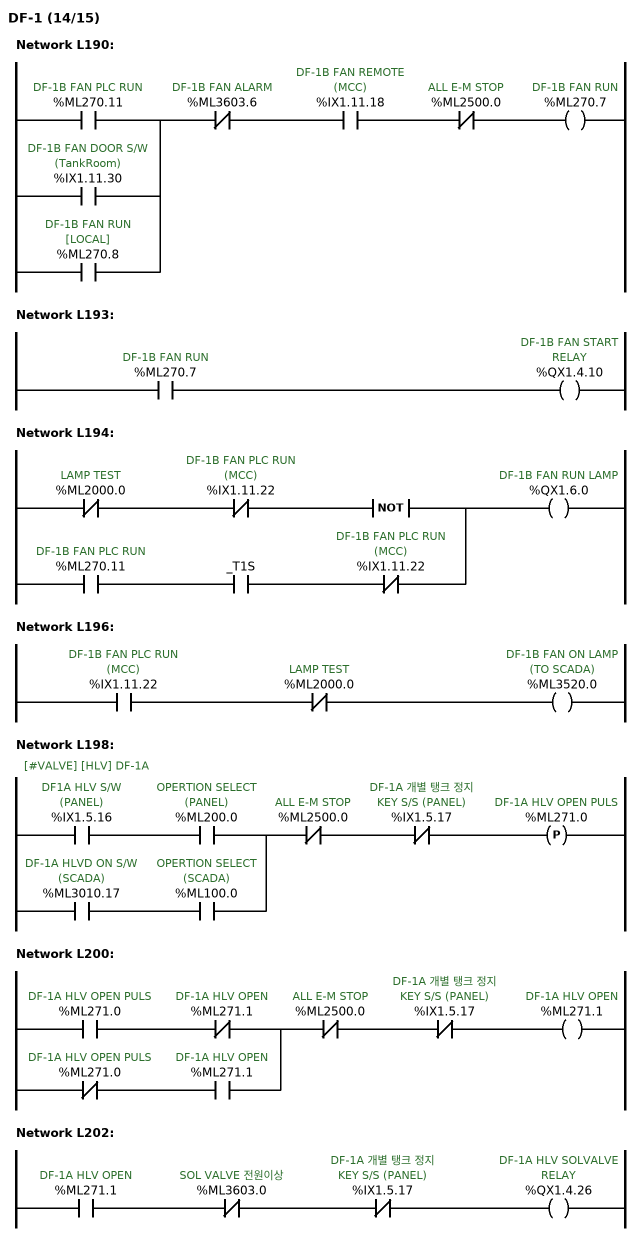
(* Rung L190 *)
%ML270.7 := (%ML270.11 OR %IX1.11.30 OR %ML270.8) AND NOT %ML3603.6 AND %IX1.11.18 AND NOT %ML2500.0;
(* Rung L193 *)
%QX1.4.10 := %ML270.7;
(* Rung L194 *)
%QX1.6.0 := NOT (NOT %ML2000.0 AND NOT %IX1.11.22) OR (%ML270.11 AND _T1S AND NOT %IX1.11.22);
(* Rung L196 *)
%ML3520.0 := %IX1.11.22 AND NOT %ML2000.0;
(* [#VALVE] [HLV] DF-1A *)
(* Rung L198 *)
_e3(CLK := ((%IX1.5.16 AND %ML200.0) OR (%ML3010.17 AND %ML100.0)) AND NOT %ML2500.0 AND NOT %IX1.5.17);
%ML271.0 := _e3.Q;
(* Rung L200 *)
%ML271.1 := ((%ML271.0 AND NOT %ML271.1) OR (NOT %ML271.0 AND %ML271.1)) AND NOT %ML2500.0 AND NOT %IX1.5.17;
(* Rung L202 *)
%QX1.4.26 := %ML271.1 AND NOT %ML3603.0 AND NOT %IX1.5.17;

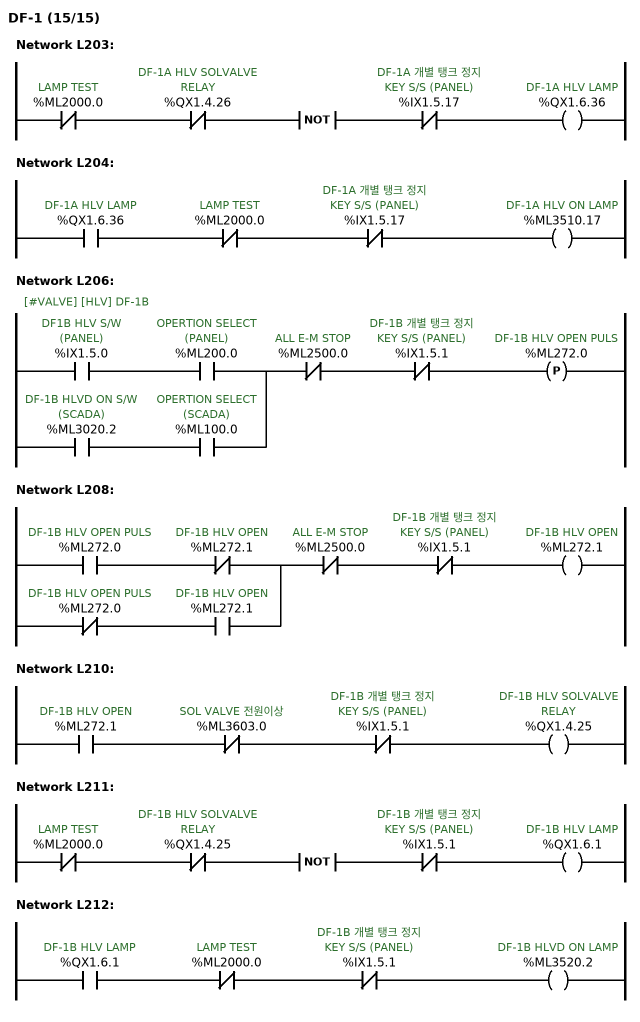
(* Rung L203 *)
%QX1.6.36 := NOT (NOT %ML2000.0 AND NOT %QX1.4.26) AND NOT %IX1.5.17;
(* Rung L204 *)
%ML3510.17 := %QX1.6.36 AND NOT %ML2000.0 AND NOT %IX1.5.17;
(* [#VALVE] [HLV] DF-1B *)
(* Rung L206 *)
_e4(CLK := ((%IX1.5.0 AND %ML200.0) OR (%ML3020.2 AND %ML100.0)) AND NOT %ML2500.0 AND NOT %IX1.5.1);
%ML272.0 := _e4.Q;
(* Rung L208 *)
%ML272.1 := ((%ML272.0 AND NOT %ML272.1) OR (NOT %ML272.0 AND %ML272.1)) AND NOT %ML2500.0 AND NOT %IX1.5.1;
(* Rung L210 *)
%QX1.4.25 := %ML272.1 AND NOT %ML3603.0 AND NOT %IX1.5.1;
(* Rung L211 *)
%QX1.6.1 := NOT (NOT %ML2000.0 AND NOT %QX1.4.25) AND NOT %IX1.5.1;
(* Rung L212 *)
%ML3520.2 := %QX1.6.1 AND NOT %ML2000.0 AND NOT %IX1.5.1;
END_PROGRAM

PROGRAM DF-M (* task: 스캔 프로그램 *)
VAR
    RP10 : TON;
    RP11 : TON;
    RP12 : TON;
    RP13 : TON;
    RP14 : TON;
    RP15 : TON;
    RP16 : TON;
    RP17 : TON;
    RP18 : TON;
    RP7 : TON;
    RP8 : TON;
    RP9 : TON;
    SUMP02 : TON; (* SP-2 *)
    SUMP04 : TON;
END_VAR
VAR
    _t1 : BOOL;
    _t2 : BOOL;
    _t3 : BOOL;
    _t4 : BOOL;
    _e5 : R_TRIG;
END_VAR

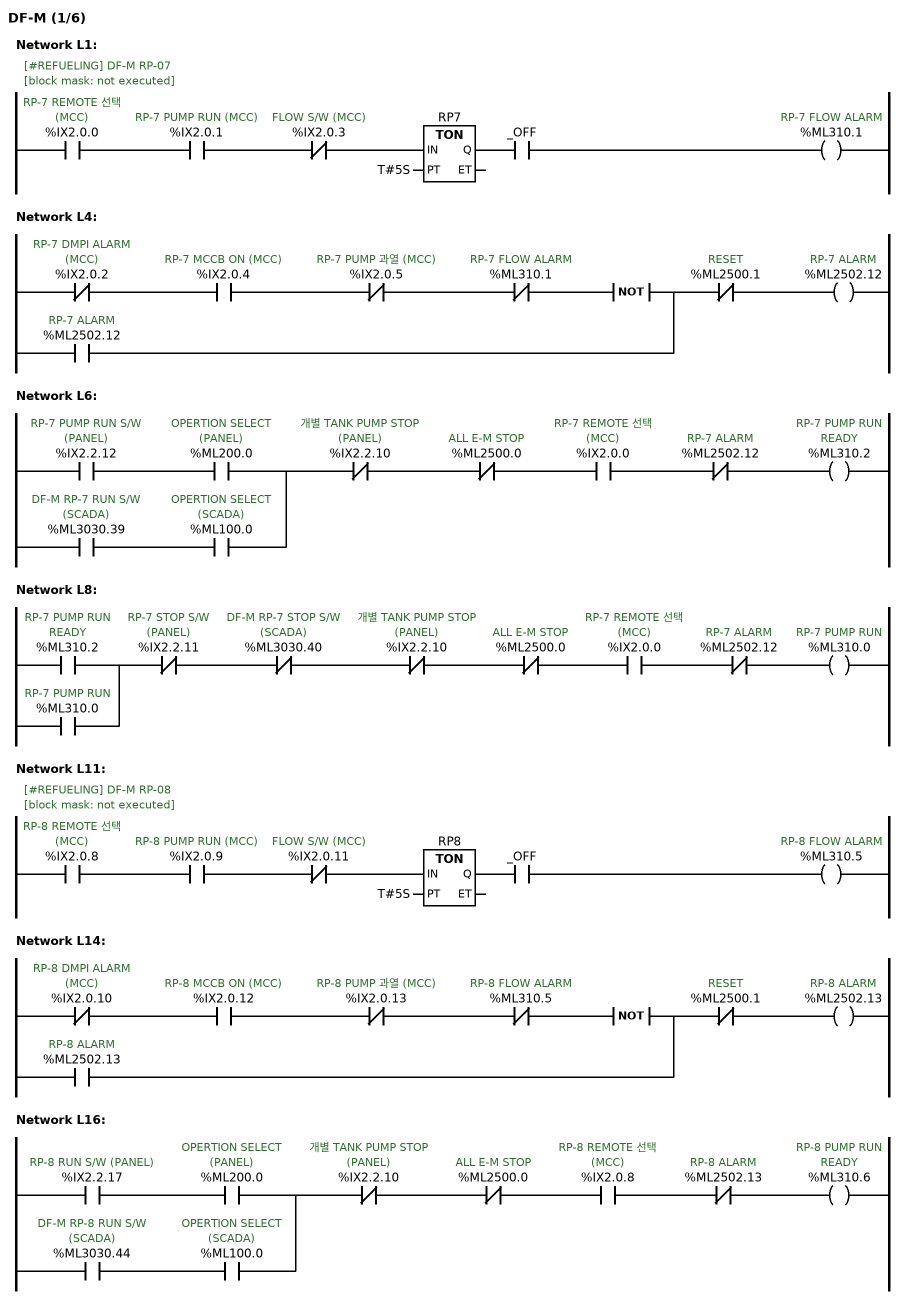
(* [#REFUELING] DF-M RP-07 *)
(* Rung L1 is block-masked: not executed *)
// RP7(IN := %IX2.0.0 AND %IX2.0.1 AND NOT %IX2.0.3, PT := T#5S);
// %ML310.1 := RP7.Q AND _OFF;
(* Rung L4 *)
%ML2502.12 := (NOT (NOT %IX2.0.2 AND %IX2.0.4 AND NOT %IX2.0.5 AND NOT %ML310.1) OR %ML2502.12) AND NOT %ML2500.1;
(* Rung L6 *)
%ML310.2 := ((%IX2.2.12 AND %ML200.0) OR (%ML3030.39 AND %ML100.0)) AND NOT %IX2.2.10 AND NOT %ML2500.0 AND %IX2.0.0 AND NOT %ML2502.12;
(* Rung L8 *)
%ML310.0 := (%ML310.2 OR %ML310.0) AND NOT %IX2.2.11 AND NOT %ML3030.40 AND NOT %IX2.2.10 AND NOT %ML2500.0 AND %IX2.0.0 AND NOT %ML2502.12;
(* [#REFUELING] DF-M RP-08 *)
(* Rung L11 is block-masked: not executed *)
// RP8(IN := %IX2.0.8 AND %IX2.0.9 AND NOT %IX2.0.11, PT := T#5S);
// %ML310.5 := RP8.Q AND _OFF;
(* Rung L14 *)
%ML2502.13 := (NOT (NOT %IX2.0.10 AND %IX2.0.12 AND NOT %IX2.0.13 AND NOT %ML310.5) OR %ML2502.13) AND NOT %ML2500.1;
(* Rung L16 *)
%ML310.6 := ((%IX2.2.17 AND %ML200.0) OR (%ML3030.44 AND %ML100.0)) AND NOT %IX2.2.10 AND NOT %ML2500.0 AND %IX2.0.8 AND NOT %ML2502.13;

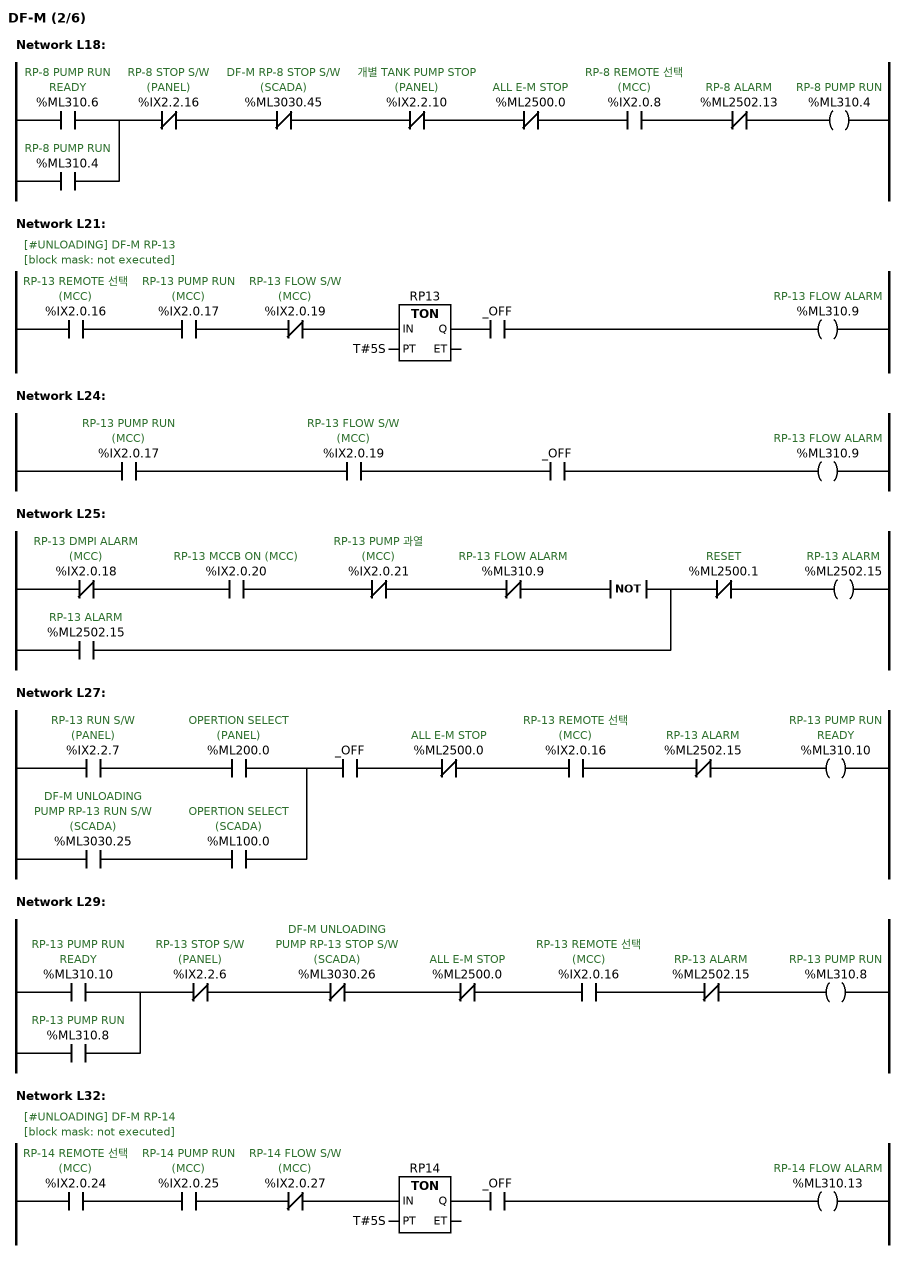
(* Rung L18 *)
%ML310.4 := (%ML310.6 OR %ML310.4) AND NOT %IX2.2.16 AND NOT %ML3030.45 AND NOT %IX2.2.10 AND NOT %ML2500.0 AND %IX2.0.8 AND NOT %ML2502.13;
(* [#UNLOADING] DF-M RP-13 *)
(* Rung L21 is block-masked: not executed *)
// RP13(IN := %IX2.0.16 AND %IX2.0.17 AND NOT %IX2.0.19, PT := T#5S);
// %ML310.9 := RP13.Q AND _OFF;
(* Rung L24 *)
%ML310.9 := %IX2.0.17 AND %IX2.0.19 AND _OFF;
(* Rung L25 *)
%ML2502.15 := (NOT (NOT %IX2.0.18 AND %IX2.0.20 AND NOT %IX2.0.21 AND NOT %ML310.9) OR %ML2502.15) AND NOT %ML2500.1;
(* Rung L27 *)
%ML310.10 := ((%IX2.2.7 AND %ML200.0) OR (%ML3030.25 AND %ML100.0)) AND _OFF AND NOT %ML2500.0 AND %IX2.0.16 AND NOT %ML2502.15;
(* Rung L29 *)
%ML310.8 := (%ML310.10 OR %ML310.8) AND NOT %IX2.2.6 AND NOT %ML3030.26 AND NOT %ML2500.0 AND %IX2.0.16 AND NOT %ML2502.15;
(* [#UNLOADING] DF-M RP-14 *)
(* Rung L32 is block-masked: not executed *)
// RP14(IN := %IX2.0.24 AND %IX2.0.25 AND NOT %IX2.0.27, PT := T#5S);
// %ML310.13 := RP14.Q AND _OFF;

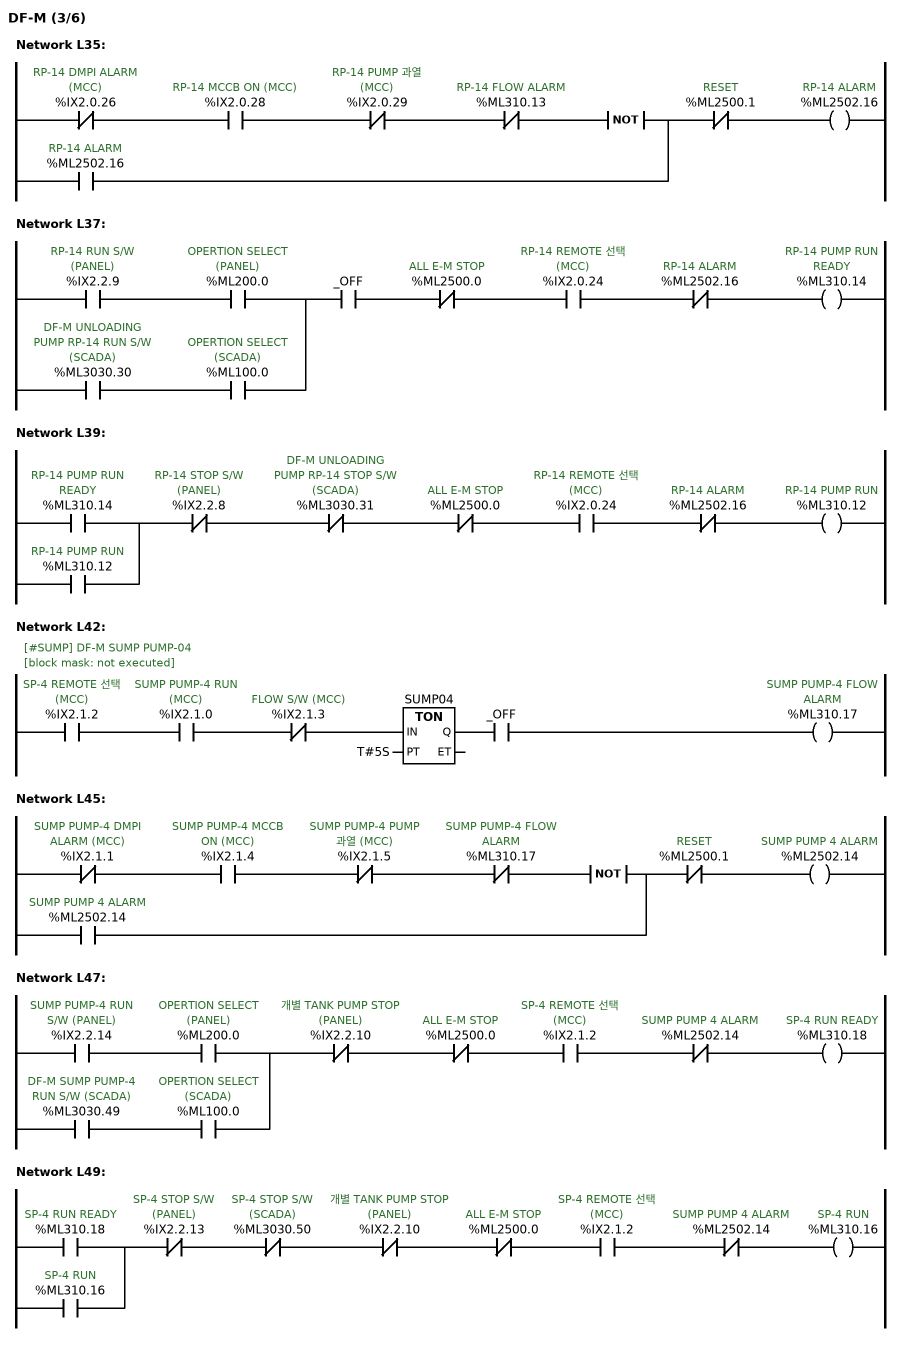
(* Rung L35 *)
%ML2502.16 := (NOT (NOT %IX2.0.26 AND %IX2.0.28 AND NOT %IX2.0.29 AND NOT %ML310.13) OR %ML2502.16) AND NOT %ML2500.1;
(* Rung L37 *)
%ML310.14 := ((%IX2.2.9 AND %ML200.0) OR (%ML3030.30 AND %ML100.0)) AND _OFF AND NOT %ML2500.0 AND %IX2.0.24 AND NOT %ML2502.16;
(* Rung L39 *)
%ML310.12 := (%ML310.14 OR %ML310.12) AND NOT %IX2.2.8 AND NOT %ML3030.31 AND NOT %ML2500.0 AND %IX2.0.24 AND NOT %ML2502.16;
(* [#SUMP] DF-M SUMP PUMP-04 *)
(* Rung L42 is block-masked: not executed *)
// SUMP04(IN := %IX2.1.2 AND %IX2.1.0 AND NOT %IX2.1.3, PT := T#5S);
// %ML310.17 := SUMP04.Q AND _OFF;
(* Rung L45 *)
%ML2502.14 := (NOT (NOT %IX2.1.1 AND %IX2.1.4 AND NOT %IX2.1.5 AND NOT %ML310.17) OR %ML2502.14) AND NOT %ML2500.1;
(* Rung L47 *)
%ML310.18 := ((%IX2.2.14 AND %ML200.0) OR (%ML3030.49 AND %ML100.0)) AND NOT %IX2.2.10 AND NOT %ML2500.0 AND %IX2.1.2 AND NOT %ML2502.14;
(* Rung L49 *)
%ML310.16 := (%ML310.18 OR %ML310.16) AND NOT %IX2.2.13 AND NOT %ML3030.50 AND NOT %IX2.2.10 AND NOT %ML2500.0 AND %IX2.1.2 AND NOT %ML2502.14;

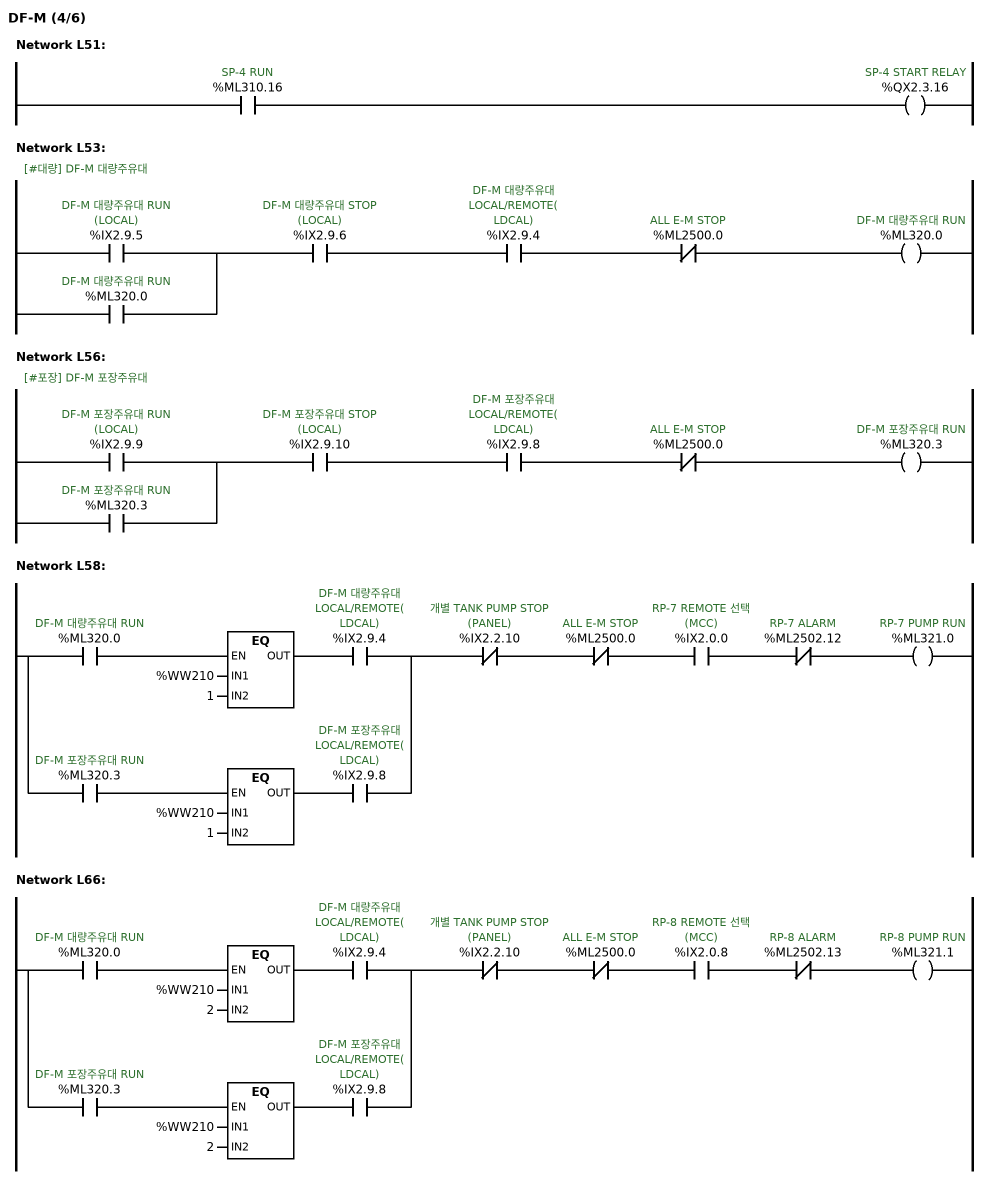
(* Rung L51 *)
%QX2.3.16 := %ML310.16;
(* [#대량] DF-M 대량주유대 *)
(* Rung L53 *)
%ML320.0 := (%IX2.9.5 OR %ML320.0) AND %IX2.9.6 AND %IX2.9.4 AND NOT %ML2500.0;
(* [#포장] DF-M 포장주유대 *)
(* Rung L56 *)
%ML320.3 := (%IX2.9.9 OR %ML320.3) AND %IX2.9.10 AND %IX2.9.8 AND NOT %ML2500.0;
(* Rung L58 *)
IF %ML320.0 THEN _t1 := %WW210 = 1; END_IF;
IF %ML320.3 THEN _t2 := %WW210 = 1; END_IF;
%ML321.0 := ((_t1 AND %IX2.9.4) OR (_t2 AND %IX2.9.8)) AND NOT %IX2.2.10 AND NOT %ML2500.0 AND %IX2.0.0 AND NOT %ML2502.12;
(* Rung L66 *)
IF %ML320.0 THEN _t3 := %WW210 = 2; END_IF;
IF %ML320.3 THEN _t4 := %WW210 = 2; END_IF;
%ML321.1 := ((_t3 AND %IX2.9.4) OR (_t4 AND %IX2.9.8)) AND NOT %IX2.2.10 AND NOT %ML2500.0 AND %IX2.0.8 AND NOT %ML2502.13;

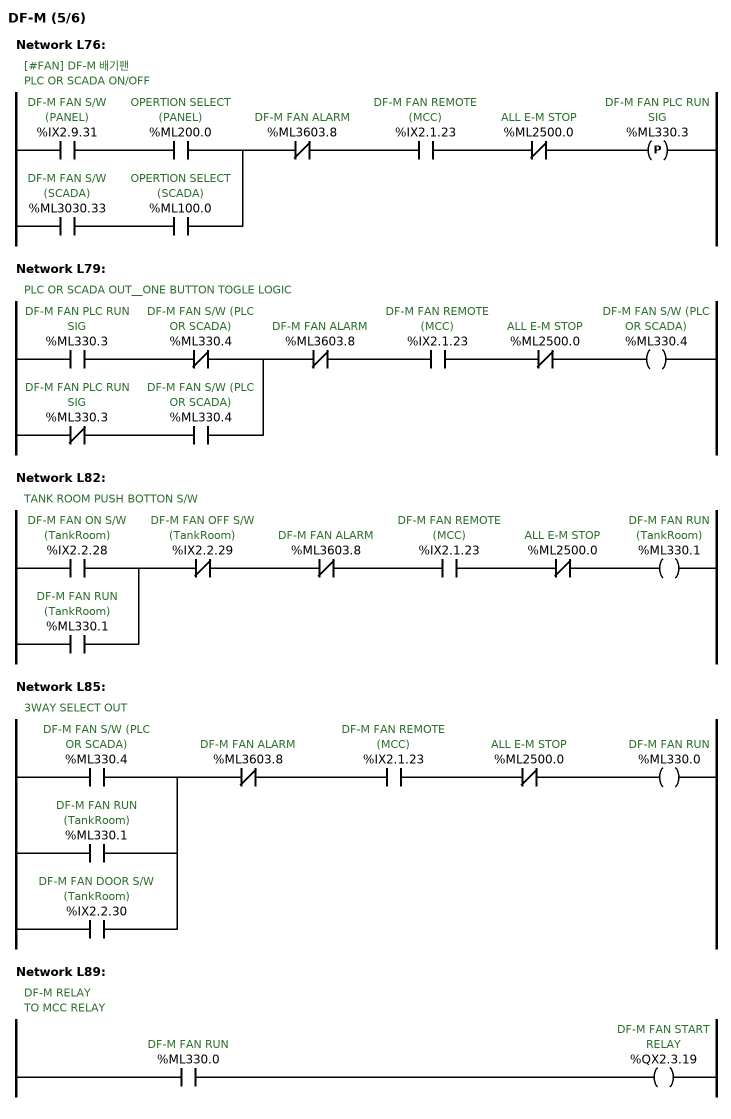
(* [#FAN] DF-M 배기팬 *)
(* PLC OR SCADA ON/OFF *)
(* Rung L76 *)
_e5(CLK := ((%IX2.9.31 AND %ML200.0) OR (%ML3030.33 AND %ML100.0)) AND NOT %ML3603.8 AND %IX2.1.23 AND NOT %ML2500.0);
%ML330.3 := _e5.Q;
(* PLC OR SCADA OUT__ONE BUTTON TOGLE LOGIC *)
(* Rung L79 *)
%ML330.4 := ((%ML330.3 AND NOT %ML330.4) OR (NOT %ML330.3 AND %ML330.4)) AND NOT %ML3603.8 AND %IX2.1.23 AND NOT %ML2500.0;
(* TANK ROOM PUSH BOTTON S/W *)
(* Rung L82 *)
%ML330.1 := (%IX2.2.28 OR %ML330.1) AND NOT %IX2.2.29 AND NOT %ML3603.8 AND %IX2.1.23 AND NOT %ML2500.0;
(* 3WAY SELECT OUT *)
(* Rung L85 *)
%ML330.0 := (%ML330.4 OR %ML330.1 OR %IX2.2.30) AND NOT %ML3603.8 AND %IX2.1.23 AND NOT %ML2500.0;
(* DF-M RELAY *)
(* Rung L89 *)
%QX2.3.19 := %ML330.0;
(* TO MCC RELAY *)

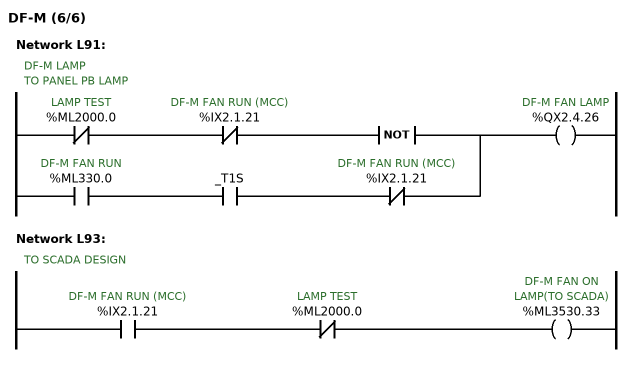
(* DF-M LAMP *)
(* Rung L91 *)
%QX2.4.26 := NOT (NOT %ML2000.0 AND NOT %IX2.1.21) OR (%ML330.0 AND _T1S AND NOT %IX2.1.21);
(* TO PANEL PB LAMP *)
(* Rung L93 *)
%ML3530.33 := %IX2.1.21 AND NOT %ML2000.0;
(* TO SCADA DESIGN *)
END_PROGRAM

PROGRAM MOGAS (* task: 스캔 프로그램 *)
VAR
    DP01 : TON; (* DRAIN PUMP FLOW SENSOR *)
    RP10 : TON;
    RP11 : TON;
    RP12 : TON;
    RP13 : TON;
    RP14 : TON;
    RP15 : TON;
    RP16 : TON;
    RP17 : TON;
    RP18 : TON;
    RP19 : TON;
    RP20 : TON;
    RP5 : TON;
    RP6 : TON;
    RP7 : TON;
    RP8 : TON;
    RP9 : TON;
    SUMP04 : TON;
END_VAR
VAR
    _t1 : BOOL;
    _t2 : BOOL;
    _t3 : BOOL;
    _t4 : BOOL;
    _e5 : R_TRIG;
END_VAR

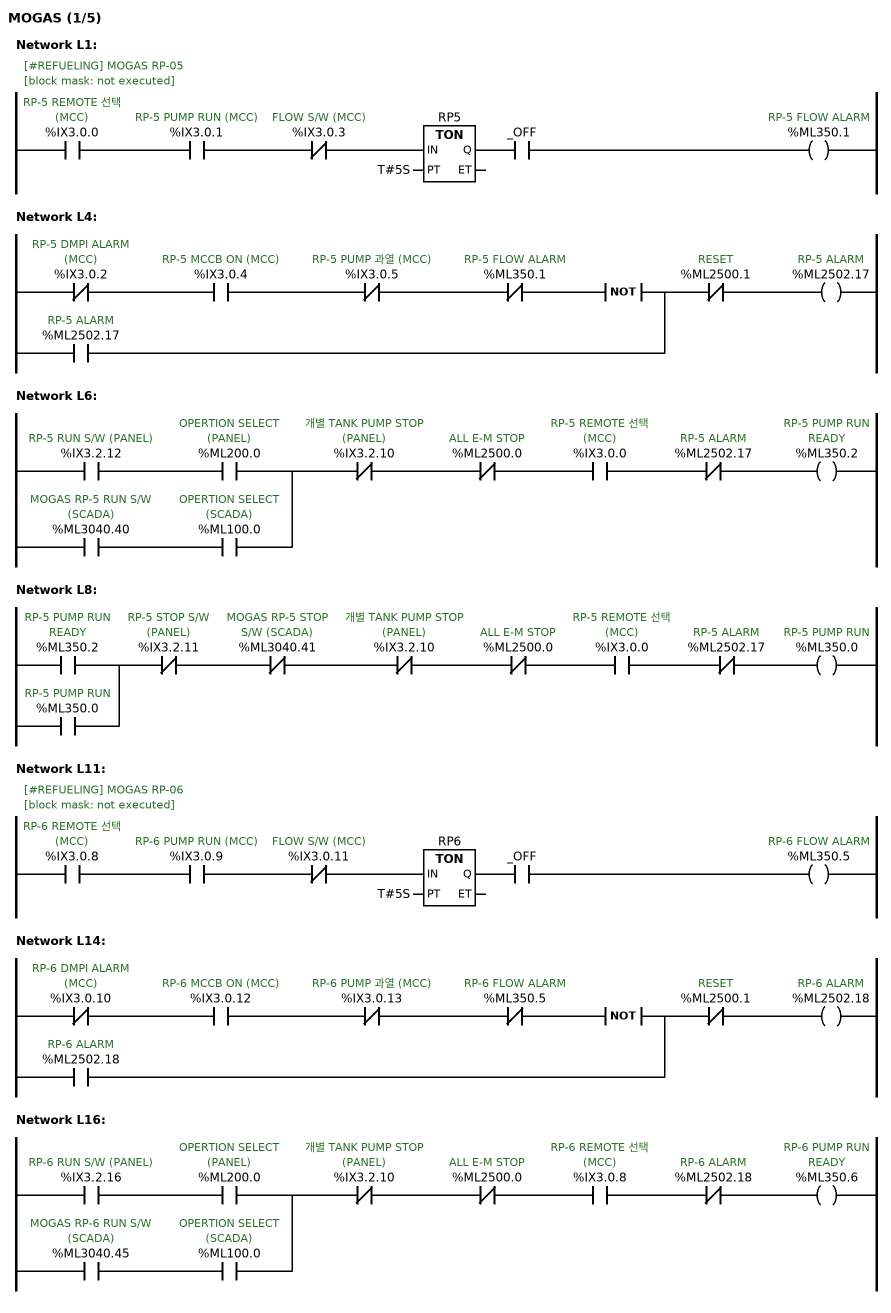
(* [#REFUELING] MOGAS RP-05 *)
(* Rung L1 is block-masked: not executed *)
// RP5(IN := %IX3.0.0 AND %IX3.0.1 AND NOT %IX3.0.3, PT := T#5S);
// %ML350.1 := RP5.Q AND _OFF;
(* Rung L4 *)
%ML2502.17 := (NOT (NOT %IX3.0.2 AND %IX3.0.4 AND NOT %IX3.0.5 AND NOT %ML350.1) OR %ML2502.17) AND NOT %ML2500.1;
(* Rung L6 *)
%ML350.2 := ((%IX3.2.12 AND %ML200.0) OR (%ML3040.40 AND %ML100.0)) AND NOT %IX3.2.10 AND NOT %ML2500.0 AND %IX3.0.0 AND NOT %ML2502.17;
(* Rung L8 *)
%ML350.0 := (%ML350.2 OR %ML350.0) AND NOT %IX3.2.11 AND NOT %ML3040.41 AND NOT %IX3.2.10 AND NOT %ML2500.0 AND %IX3.0.0 AND NOT %ML2502.17;
(* [#REFUELING] MOGAS RP-06 *)
(* Rung L11 is block-masked: not executed *)
// RP6(IN := %IX3.0.8 AND %IX3.0.9 AND NOT %IX3.0.11, PT := T#5S);
// %ML350.5 := RP6.Q AND _OFF;
(* Rung L14 *)
%ML2502.18 := (NOT (NOT %IX3.0.10 AND %IX3.0.12 AND NOT %IX3.0.13 AND NOT %ML350.5) OR %ML2502.18) AND NOT %ML2500.1;
(* Rung L16 *)
%ML350.6 := ((%IX3.2.16 AND %ML200.0) OR (%ML3040.45 AND %ML100.0)) AND NOT %IX3.2.10 AND NOT %ML2500.0 AND %IX3.0.8 AND NOT %ML2502.18;

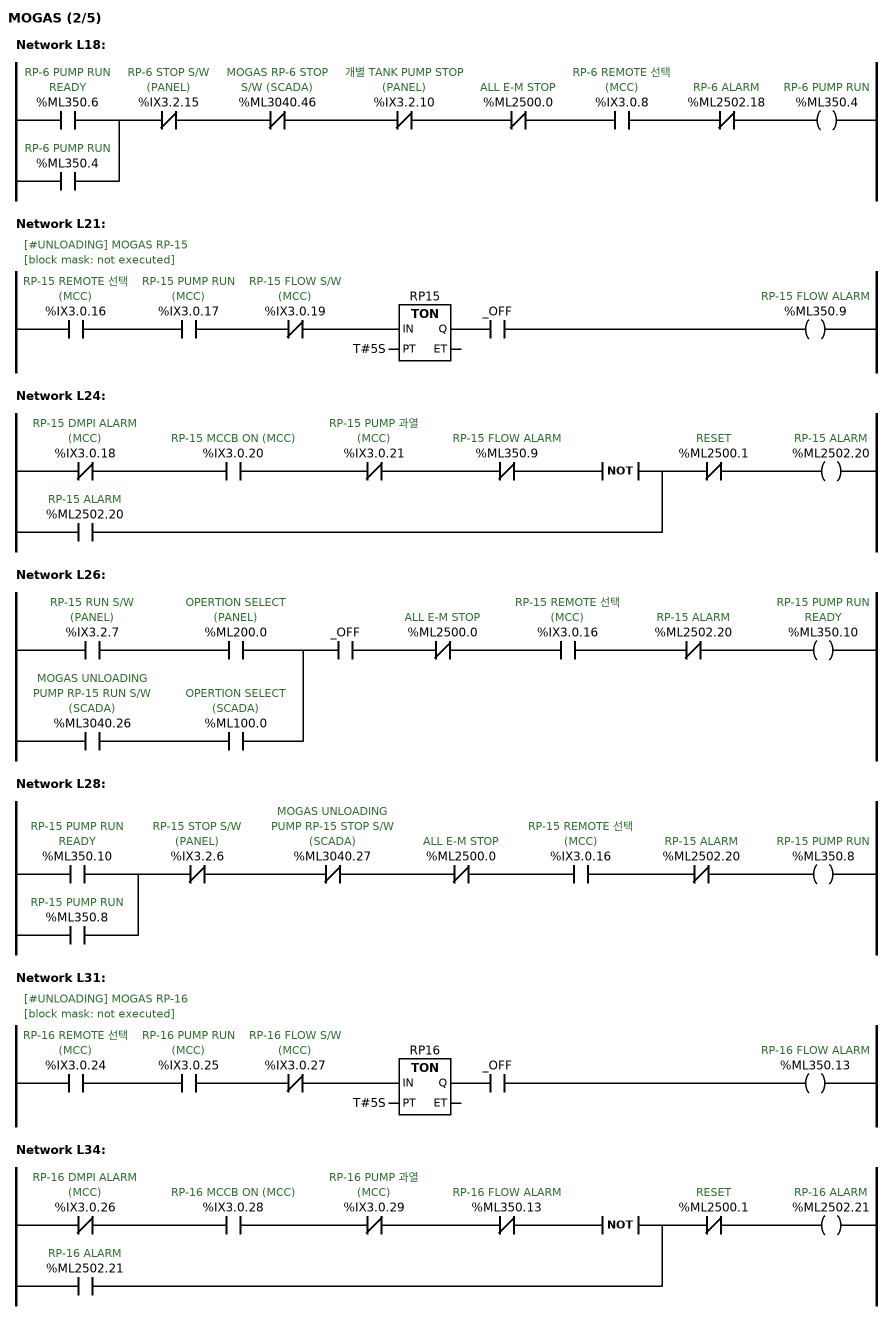
(* Rung L18 *)
%ML350.4 := (%ML350.6 OR %ML350.4) AND NOT %IX3.2.15 AND NOT %ML3040.46 AND NOT %IX3.2.10 AND NOT %ML2500.0 AND %IX3.0.8 AND NOT %ML2502.18;
(* [#UNLOADING] MOGAS RP-15 *)
(* Rung L21 is block-masked: not executed *)
// RP15(IN := %IX3.0.16 AND %IX3.0.17 AND NOT %IX3.0.19, PT := T#5S);
// %ML350.9 := RP15.Q AND _OFF;
(* Rung L24 *)
%ML2502.20 := (NOT (NOT %IX3.0.18 AND %IX3.0.20 AND NOT %IX3.0.21 AND NOT %ML350.9) OR %ML2502.20) AND NOT %ML2500.1;
(* Rung L26 *)
%ML350.10 := ((%IX3.2.7 AND %ML200.0) OR (%ML3040.26 AND %ML100.0)) AND _OFF AND NOT %ML2500.0 AND %IX3.0.16 AND NOT %ML2502.20;
(* Rung L28 *)
%ML350.8 := (%ML350.10 OR %ML350.8) AND NOT %IX3.2.6 AND NOT %ML3040.27 AND NOT %ML2500.0 AND %IX3.0.16 AND NOT %ML2502.20;
(* [#UNLOADING] MOGAS RP-16 *)
(* Rung L31 is block-masked: not executed *)
// RP16(IN := %IX3.0.24 AND %IX3.0.25 AND NOT %IX3.0.27, PT := T#5S);
// %ML350.13 := RP16.Q AND _OFF;
(* Rung L34 *)
%ML2502.21 := (NOT (NOT %IX3.0.26 AND %IX3.0.28 AND NOT %IX3.0.29 AND NOT %ML350.13) OR %ML2502.21) AND NOT %ML2500.1;

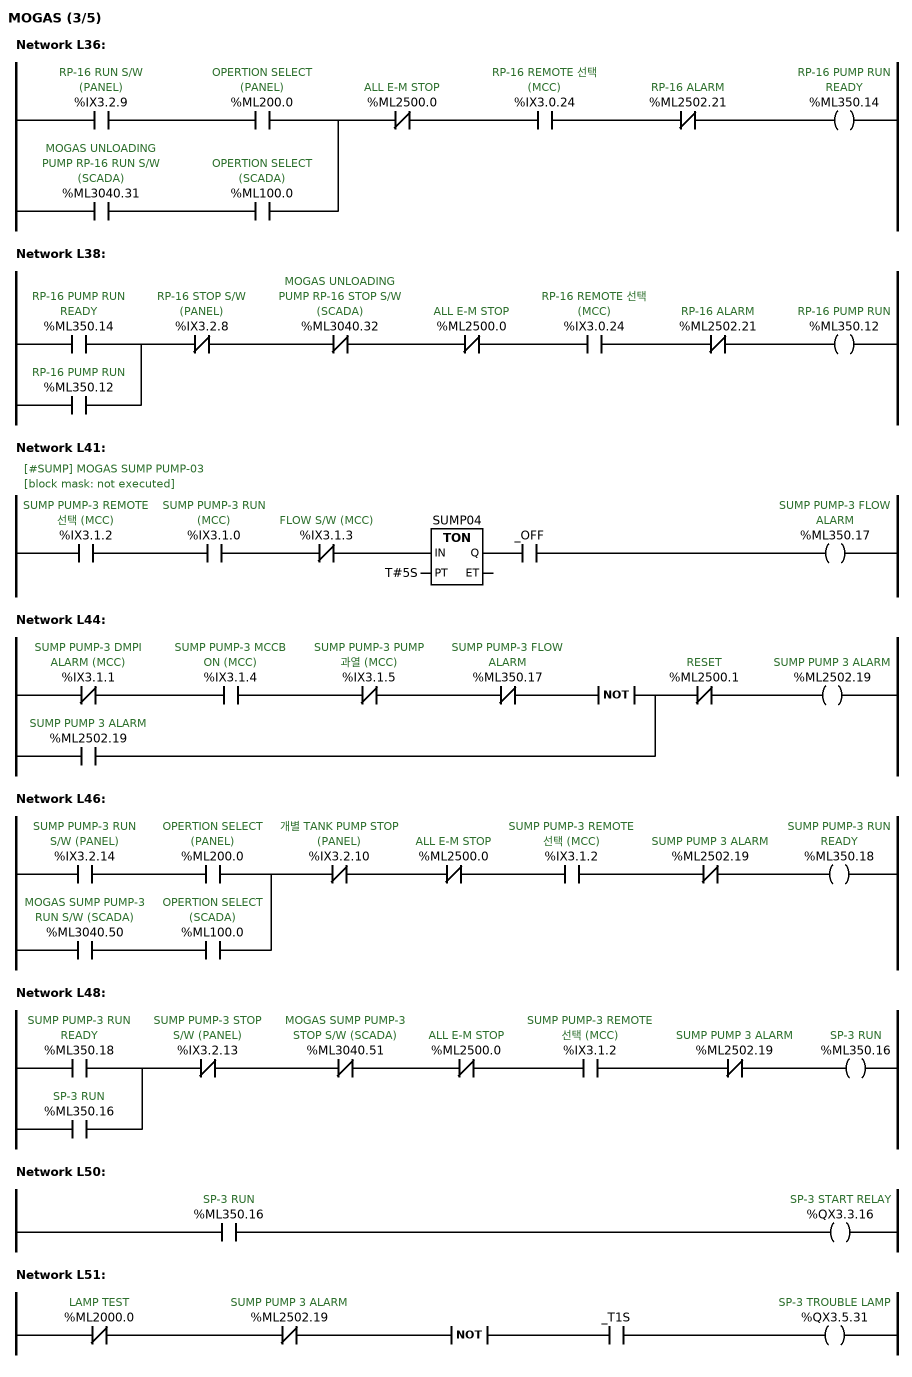
(* Rung L36 *)
%ML350.14 := ((%IX3.2.9 AND %ML200.0) OR (%ML3040.31 AND %ML100.0)) AND NOT %ML2500.0 AND %IX3.0.24 AND NOT %ML2502.21;
(* Rung L38 *)
%ML350.12 := (%ML350.14 OR %ML350.12) AND NOT %IX3.2.8 AND NOT %ML3040.32 AND NOT %ML2500.0 AND %IX3.0.24 AND NOT %ML2502.21;
(* [#SUMP] MOGAS SUMP PUMP-03 *)
(* Rung L41 is block-masked: not executed *)
// SUMP04(IN := %IX3.1.2 AND %IX3.1.0 AND NOT %IX3.1.3, PT := T#5S);
// %ML350.17 := SUMP04.Q AND _OFF;
(* Rung L44 *)
%ML2502.19 := (NOT (NOT %IX3.1.1 AND %IX3.1.4 AND NOT %IX3.1.5 AND NOT %ML350.17) OR %ML2502.19) AND NOT %ML2500.1;
(* Rung L46 *)
%ML350.18 := ((%IX3.2.14 AND %ML200.0) OR (%ML3040.50 AND %ML100.0)) AND NOT %IX3.2.10 AND NOT %ML2500.0 AND %IX3.1.2 AND NOT %ML2502.19;
(* Rung L48 *)
%ML350.16 := (%ML350.18 OR %ML350.16) AND NOT %IX3.2.13 AND NOT %ML3040.51 AND NOT %ML2500.0 AND %IX3.1.2 AND NOT %ML2502.19;
(* Rung L50 *)
%QX3.3.16 := %ML350.16;
(* Rung L51 *)
%QX3.5.31 := NOT (NOT %ML2000.0 AND NOT %ML2502.19) AND _T1S;

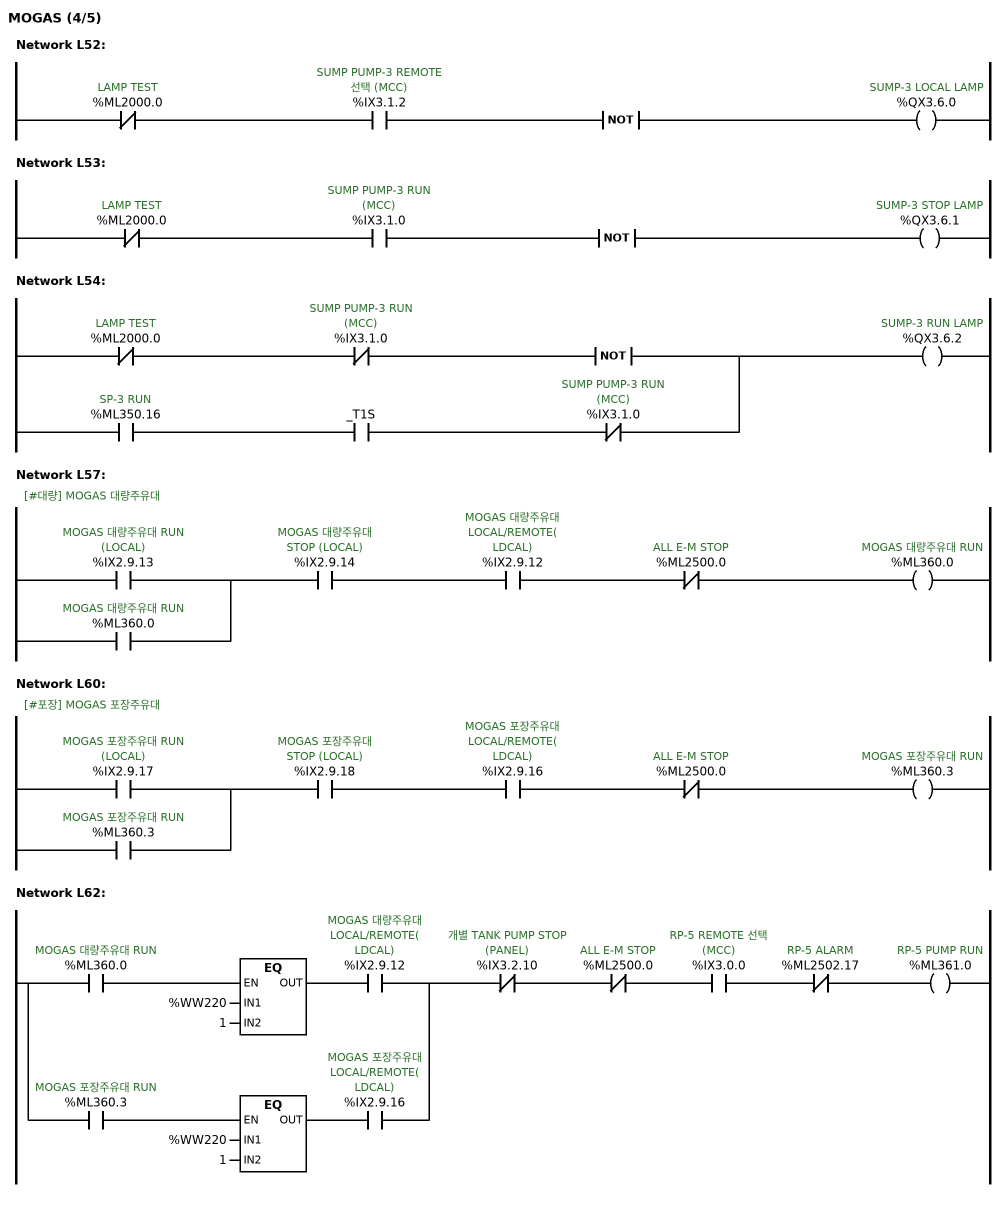
(* Rung L52 *)
%QX3.6.0 := NOT (NOT %ML2000.0 AND %IX3.1.2);
(* Rung L53 *)
%QX3.6.1 := NOT (NOT %ML2000.0 AND %IX3.1.0);
(* Rung L54 *)
%QX3.6.2 := NOT (NOT %ML2000.0 AND NOT %IX3.1.0) OR (%ML350.16 AND _T1S AND NOT %IX3.1.0);
(* [#대량] MOGAS 대량주유대 *)
(* Rung L57 *)
%ML360.0 := (%IX2.9.13 OR %ML360.0) AND %IX2.9.14 AND %IX2.9.12 AND NOT %ML2500.0;
(* [#포장] MOGAS 포장주유대 *)
(* Rung L60 *)
%ML360.3 := (%IX2.9.17 OR %ML360.3) AND %IX2.9.18 AND %IX2.9.16 AND NOT %ML2500.0;
(* Rung L62 *)
IF %ML360.0 THEN _t1 := %WW220 = 1; END_IF;
IF %ML360.3 THEN _t2 := %WW220 = 1; END_IF;
%ML361.0 := ((_t1 AND %IX2.9.12) OR (_t2 AND %IX2.9.16)) AND NOT %IX3.2.10 AND NOT %ML2500.0 AND %IX3.0.0 AND NOT %ML2502.17;

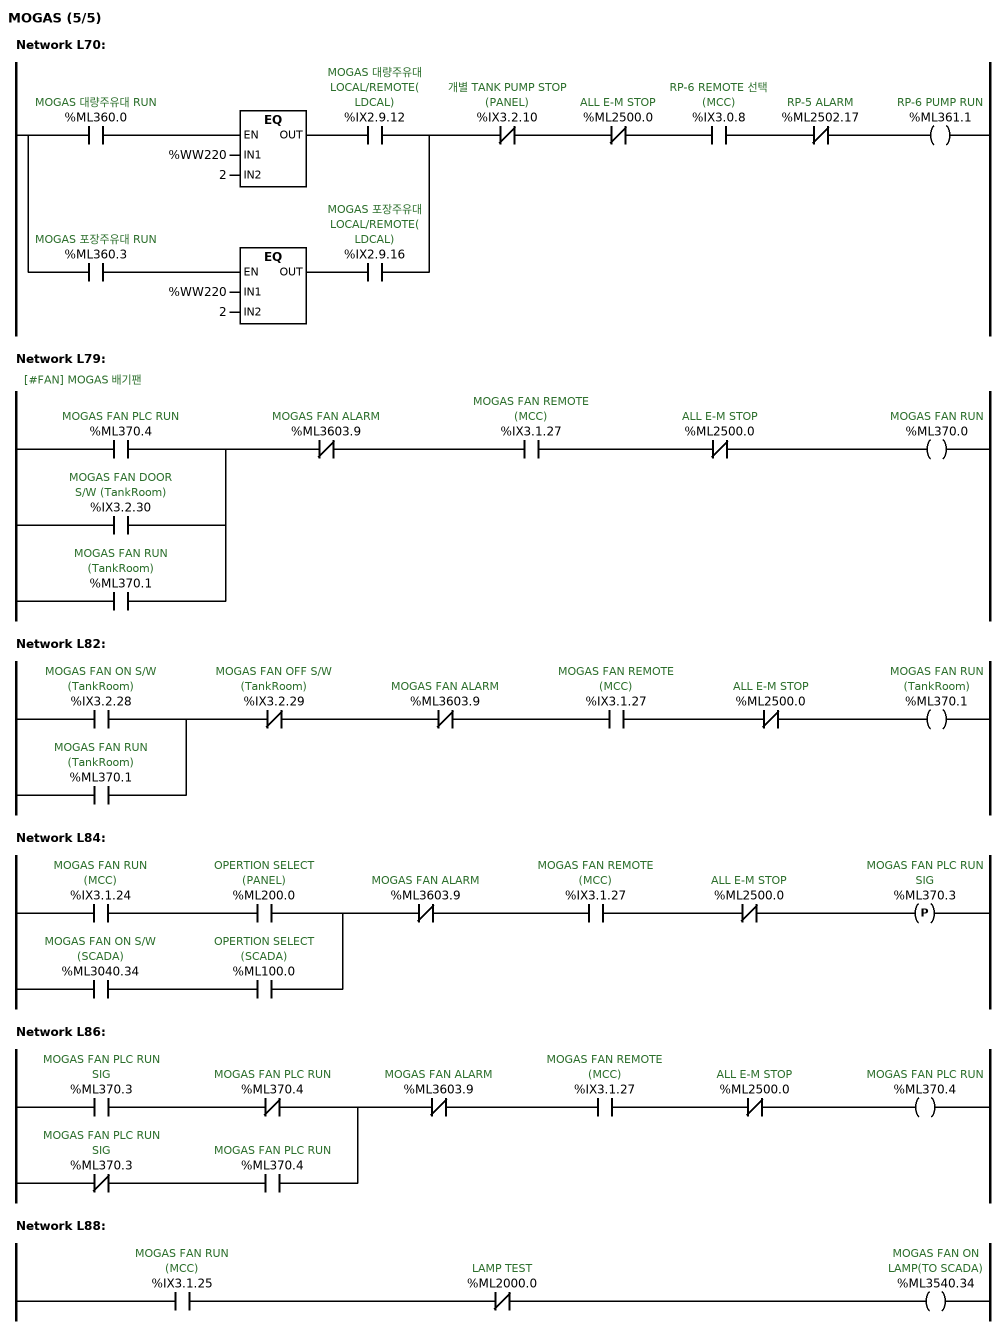
(* Rung L70 *)
IF %ML360.0 THEN _t3 := %WW220 = 2; END_IF;
IF %ML360.3 THEN _t4 := %WW220 = 2; END_IF;
%ML361.1 := ((_t3 AND %IX2.9.12) OR (_t4 AND %IX2.9.16)) AND NOT %IX3.2.10 AND NOT %ML2500.0 AND %IX3.0.8 AND NOT %ML2502.17;
(* [#FAN] MOGAS 배기팬 *)
(* Rung L79 *)
%ML370.0 := (%ML370.4 OR %IX3.2.30 OR %ML370.1) AND NOT %ML3603.9 AND %IX3.1.27 AND NOT %ML2500.0;
(* Rung L82 *)
%ML370.1 := (%IX3.2.28 OR %ML370.1) AND NOT %IX3.2.29 AND NOT %ML3603.9 AND %IX3.1.27 AND NOT %ML2500.0;
(* Rung L84 *)
_e5(CLK := ((%IX3.1.24 AND %ML200.0) OR (%ML3040.34 AND %ML100.0)) AND NOT %ML3603.9 AND %IX3.1.27 AND NOT %ML2500.0);
%ML370.3 := _e5.Q;
(* Rung L86 *)
%ML370.4 := ((%ML370.3 AND NOT %ML370.4) OR (NOT %ML370.3 AND %ML370.4)) AND NOT %ML3603.9 AND %IX3.1.27 AND NOT %ML2500.0;
(* Rung L88 *)
%ML3540.34 := %IX3.1.25 AND NOT %ML2000.0;
END_PROGRAM

PROGRAM ANALOGUE (* task: 스캔 프로그램 *)
VAR
    DF1A_LEVEL_PER : INT;
    DF1B_LEVEL_PER : INT;
    DFM_LEVEL_PER : INT;
    DTK1_LEVEL_PER : INT;
    DTK2_LEVEL_PER : INT;
    FIT_1 : INT;
    FIT_2 : INT;
    MOGAS_LEVEL_PER : INT;
END_VAR
VAR_EXTERNAL
    _0108_CH0_ACT : BOOL; (* AT %UX1.8.16 *) (* 절연형 아날로그입력 모듈: 채널0 운전중 *)
    _0108_CH0_DATA : INT; (* AT %UW1.8.2 *) (* 절연형 아날로그입력 모듈: 채널0 변환값 *)
    _0108_CH0_IDD : BOOL; (* AT %UX1.8.160 *) (* 절연형 아날로그입력 모듈: 채널0 입력단선검출 *)
    _0108_CH1_ACT : BOOL; (* AT %UX1.8.17 *) (* 절연형 아날로그입력 모듈: 채널1 운전중 *)
    _0108_CH1_DATA : INT; (* AT %UW1.8.3 *) (* 절연형 아날로그입력 모듈: 채널1 변환값 *)
    _0108_CH1_IDD : BOOL; (* AT %UX1.8.161 *) (* 절연형 아날로그입력 모듈: 채널1 입력단선검출 *)
    _0108_CH2_ACT : BOOL; (* AT %UX1.8.18 *) (* 절연형 아날로그입력 모듈: 채널2 운전중 *)
    _0108_CH2_DATA : INT; (* AT %UW1.8.4 *) (* 절연형 아날로그입력 모듈: 채널2 변환값 *)
    _0108_CH2_IDD : BOOL; (* AT %UX1.8.162 *) (* 절연형 아날로그입력 모듈: 채널2 입력단선검출 *)
    _0108_CH3_ACT : BOOL; (* AT %UX1.8.19 *) (* 절연형 아날로그입력 모듈: 채널3 운전중 *)
    _0108_CH3_DATA : INT; (* AT %UW1.8.5 *) (* 절연형 아날로그입력 모듈: 채널3 변환값 *)
    _0108_CH3_IDD : BOOL; (* AT %UX1.8.163 *) (* 절연형 아날로그입력 모듈: 채널3 입력단선검출 *)
    _0109_CH0_ACT : BOOL; (* AT %UX1.9.16 *) (* 절연형 아날로그출력 모듈: 채널0 운전중 *)
    _0109_CH0_DATA : INT; (* AT %UW1.9.3 *) (* 절연형 아날로그출력 모듈: 채널0 입력값 *)
    _0109_CH0_ERR : BOOL; (* AT %UX1.9.0 *) (* 절연형 아날로그출력 모듈: 채널0 에러 *)
    _0109_CH0_OUTEN : BOOL; (* AT %UX1.9.32 *) (* 절연형 아날로그출력 모듈: 채널0 출력상태설정 *)
    _0109_CH1_ACT : BOOL; (* AT %UX1.9.17 *) (* 절연형 아날로그출력 모듈: 채널1 운전중 *)
    _0109_CH1_DATA : INT; (* AT %UW1.9.4 *) (* 절연형 아날로그출력 모듈: 채널1 입력값 *)
    _0109_CH1_ERR : BOOL; (* AT %UX1.9.1 *) (* 절연형 아날로그출력 모듈: 채널1 에러 *)
    _0109_CH2_ACT : BOOL; (* AT %UX1.9.18 *) (* 절연형 아날로그출력 모듈: 채널2 운전중 *)
    _0109_CH2_DATA : INT; (* AT %UW1.9.5 *) (* 절연형 아날로그출력 모듈: 채널2 입력값 *)
    _0109_CH2_ERR : BOOL; (* AT %UX1.9.2 *) (* 절연형 아날로그출력 모듈: 채널2 에러 *)
    _0109_CH3_ACT : BOOL; (* AT %UX1.9.19 *) (* 절연형 아날로그출력 모듈: 채널3 운전중 *)
    _0109_CH3_DATA : INT; (* AT %UW1.9.6 *) (* 절연형 아날로그출력 모듈: 채널3 입력값 *)
    _0109_CH3_ERR : BOOL; (* AT %UX1.9.3 *) (* 절연형 아날로그출력 모듈: 채널3 에러 *)
    _0109_OUTEN : WORD; (* AT %UW1.9.2 *) (* 절연형 아날로그출력 모듈: 출력상태 설정 *)
    _0110_CH0_ACT : BOOL; (* AT %UX1.10.16 *) (* 절연형 아날로그출력 모듈: 채널0 운전중 *)
    _0110_CH0_DATA : INT; (* AT %UW1.10.3 *) (* 절연형 아날로그출력 모듈: 채널0 입력값 *)
    _0110_CH0_ERR : BOOL; (* AT %UX1.10.0 *) (* 절연형 아날로그출력 모듈: 채널0 에러 *)
    _0110_OUTEN : WORD; (* AT %UW1.10.2 *) (* 절연형 아날로그출력 모듈: 출력상태 설정 *)
    _0206_CH0_ACT : BOOL; (* AT %UX2.6.16 *) (* 절연형 아날로그입력 모듈: 채널0 운전중 *)
    _0206_CH0_DATA : INT; (* AT %UW2.6.2 *) (* 절연형 아날로그입력 모듈: 채널0 변환값 *)
    _0206_CH0_IDD : BOOL; (* AT %UX2.6.160 *) (* 절연형 아날로그입력 모듈: 채널0 입력단선검출 *)
    _0206_CH1_ACT : BOOL; (* AT %UX2.6.17 *) (* 절연형 아날로그입력 모듈: 채널1 운전중 *)
    _0206_CH1_DATA : INT; (* AT %UW2.6.3 *) (* 절연형 아날로그입력 모듈: 채널1 변환값 *)
    _0206_CH1_IDD : BOOL; (* AT %UX2.6.161 *) (* 절연형 아날로그입력 모듈: 채널1 입력단선검출 *)
    _0206_CH2_ACT : BOOL; (* AT %UX2.6.18 *) (* 절연형 아날로그입력 모듈: 채널2 운전중 *)
    _0206_CH2_DATA : INT; (* AT %UW2.6.4 *) (* 절연형 아날로그입력 모듈: 채널2 변환값 *)
    _0206_CH2_IDD : BOOL; (* AT %UX2.6.162 *) (* 절연형 아날로그입력 모듈: 채널2 입력단선검출 *)
    _0206_CH3_ACT : BOOL; (* AT %UX2.6.19 *) (* 절연형 아날로그입력 모듈: 채널3 운전중 *)
    _0206_CH3_DATA : INT; (* AT %UW2.6.5 *) (* 절연형 아날로그입력 모듈: 채널3 변환값 *)
    _0206_CH3_IDD : BOOL; (* AT %UX2.6.163 *) (* 절연형 아날로그입력 모듈: 채널3 입력단선검출 *)
    _0207_CH0_ACT : BOOL; (* AT %UX2.7.16 *) (* 절연형 아날로그출력 모듈: 채널0 운전중 *)
    _0207_CH0_DATA : INT; (* AT %UW2.7.3 *) (* 절연형 아날로그출력 모듈: 채널0 입력값 *)
    _0207_CH0_ERR : BOOL; (* AT %UX2.7.0 *) (* 절연형 아날로그출력 모듈: 채널0 에러 *)
    _0207_CH1_ACT : BOOL; (* AT %UX2.7.17 *) (* 절연형 아날로그출력 모듈: 채널1 운전중 *)
    _0207_CH1_DATA : INT; (* AT %UW2.7.4 *) (* 절연형 아날로그출력 모듈: 채널1 입력값 *)
    _0207_CH2_ACT : BOOL; (* AT %UX2.7.18 *) (* 절연형 아날로그출력 모듈: 채널2 운전중 *)
    _0207_CH2_DATA : INT; (* AT %UW2.7.5 *) (* 절연형 아날로그출력 모듈: 채널2 입력값 *)
    _0207_CH2_ERR : BOOL; (* AT %UX2.7.2 *) (* 절연형 아날로그출력 모듈: 채널2 에러 *)
    _0207_CH3_DATA : INT; (* AT %UW2.7.6 *) (* 절연형 아날로그출력 모듈: 채널3 입력값 *)
    _0207_OUTEN : WORD; (* AT %UW2.7.2 *) (* 절연형 아날로그출력 모듈: 출력상태 설정 *)
    _0307_CH0_ACT : BOOL; (* AT %UX3.7.16 *) (* 절연형 아날로그입력 모듈: 채널0 운전중 *)
    _0307_CH0_DATA : INT; (* AT %UW3.7.2 *) (* 절연형 아날로그입력 모듈: 채널0 변환값 *)
    _0307_CH0_IDD : BOOL; (* AT %UX3.7.160 *) (* 절연형 아날로그입력 모듈: 채널0 입력단선검출 *)
    _0307_CH1_ACT : BOOL; (* AT %UX3.7.17 *) (* 절연형 아날로그입력 모듈: 채널1 운전중 *)
    _0307_CH1_DATA : INT; (* AT %UW3.7.3 *) (* 절연형 아날로그입력 모듈: 채널1 변환값 *)
    _0307_CH1_IDD : BOOL; (* AT %UX3.7.161 *) (* 절연형 아날로그입력 모듈: 채널1 입력단선검출 *)
    _0307_CH2_ACT : BOOL; (* AT %UX3.7.18 *) (* 절연형 아날로그입력 모듈: 채널2 운전중 *)
    _0307_CH2_DATA : INT; (* AT %UW3.7.4 *) (* 절연형 아날로그입력 모듈: 채널2 변환값 *)
    _0307_CH2_IDD : BOOL; (* AT %UX3.7.162 *) (* 절연형 아날로그입력 모듈: 채널2 입력단선검출 *)
    _0307_CH3_DATA : INT; (* AT %UW3.7.5 *) (* 절연형 아날로그입력 모듈: 채널3 변환값 *)
    _0307_CH3_IDD : BOOL; (* AT %UX3.7.163 *) (* 절연형 아날로그입력 모듈: 채널3 입력단선검출 *)
    _0308_CH0_ACT : BOOL; (* AT %UX3.8.16 *) (* 절연형 아날로그출력 모듈: 채널0 운전중 *)
    _0308_CH0_DATA : INT; (* AT %UW3.8.3 *) (* 절연형 아날로그출력 모듈: 채널0 입력값 *)
    _0308_CH1_ACT : BOOL; (* AT %UX3.8.17 *) (* 절연형 아날로그출력 모듈: 채널1 운전중 *)
    _0308_CH1_DATA : INT; (* AT %UW3.8.4 *) (* 절연형 아날로그출력 모듈: 채널1 입력값 *)
    _0308_CH2_ACT : BOOL; (* AT %UX3.8.18 *) (* 절연형 아날로그출력 모듈: 채널2 운전중 *)
    _0308_CH2_DATA : INT; (* AT %UW3.8.5 *) (* 절연형 아날로그출력 모듈: 채널2 입력값 *)
    _0308_CH2_ERR : BOOL; (* AT %UX3.8.2 *) (* 절연형 아날로그출력 모듈: 채널2 에러 *)
    _0308_CH3_ACT : BOOL; (* AT %UX3.8.19 *) (* 절연형 아날로그출력 모듈: 채널3 운전중 *)
    _0308_CH3_DATA : INT; (* AT %UW3.8.6 *) (* 절연형 아날로그출력 모듈: 채널3 입력값 *)
    _0308_CH3_ERR : BOOL; (* AT %UX3.8.3 *) (* 절연형 아날로그출력 모듈: 채널3 에러 *)
    _0308_OUTEN : WORD; (* AT %UW3.8.2 *) (* 절연형 아날로그출력 모듈: 출력상태 설정 *)
END_VAR
VAR_EXTERNAL CONSTANT
    _F0308_CH0_DEC_RATE : UINT; (* 절연형 아날로그출력 모듈: 채널0 변화율 감소값 *)
    _F0308_CH0_STAT : UINT; (* 절연형 아날로그출력 모듈: 채널0 이상 상태 출력 설정값 *)
    _F0308_LIMIT_EN : UINT; (* 절연형 아날로그출력 모듈: 출력제한 채널 설정 *)
END_VAR
VAR
    _t1 : BOOL;
    _t2 : BOOL;
    _t3 : BOOL;
    _t4 : BOOL;
    _t5 : BOOL;
    _t6 : BOOL;
    _t7 : BOOL;
    _t8 : BOOL;
    _t9 : BOOL;
    _t10 : BOOL;
    _t11 : BOOL;
    _t12 : BOOL;
    _t13 : BOOL;
END_VAR

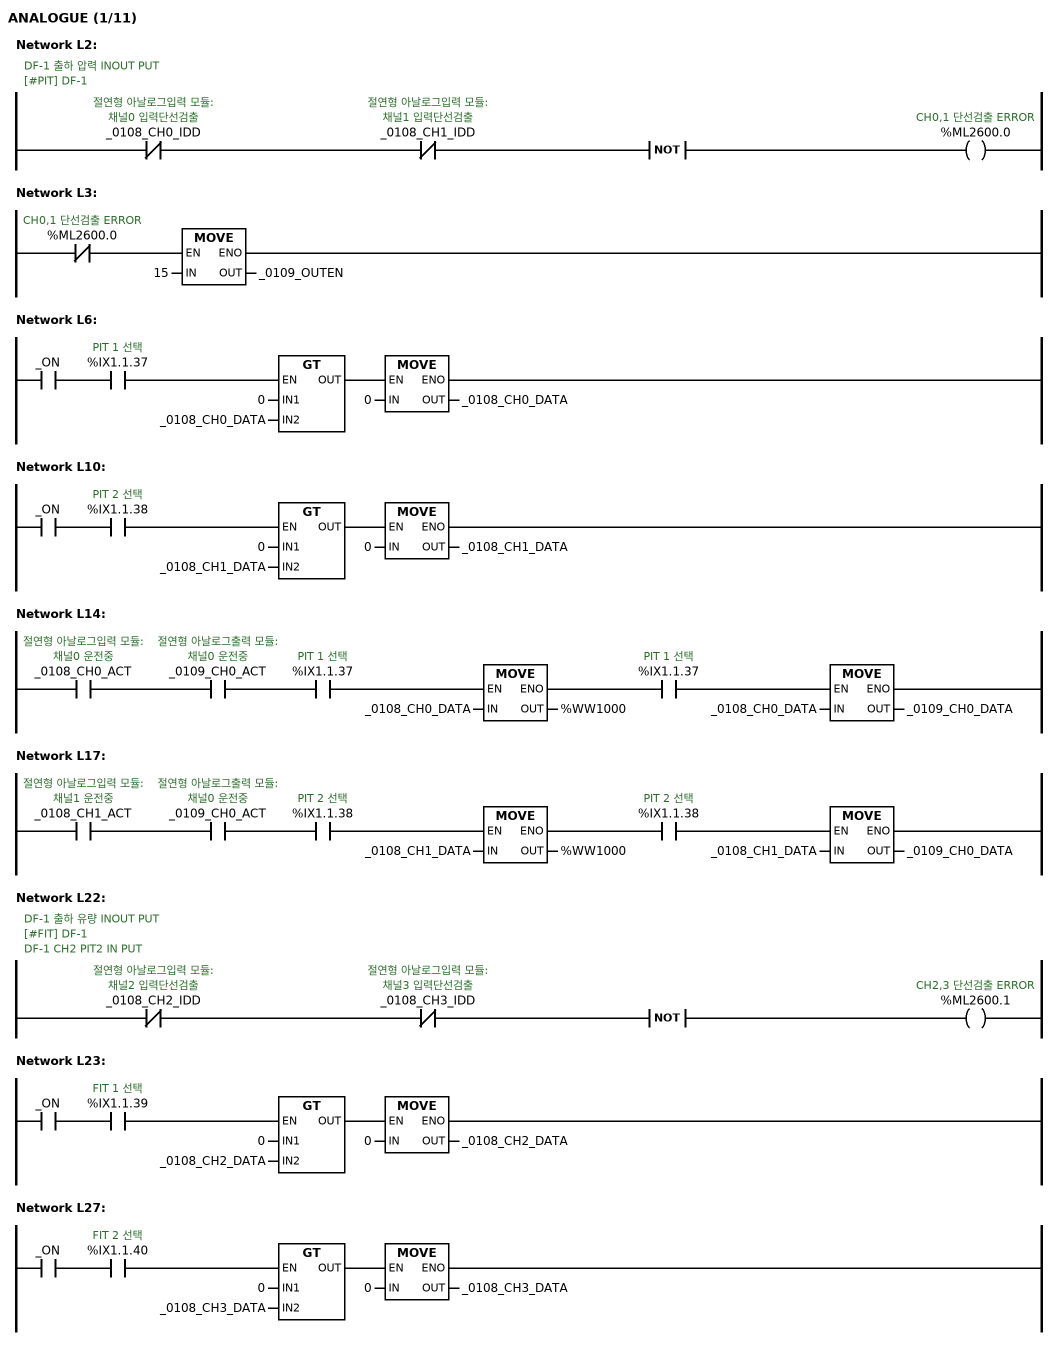
(* DF-1 출하 압력 INOUT PUT *)
(* [#PIT] DF-1 *)
(* Rung L2 *)
%ML2600.0 := NOT (NOT _0108_CH0_IDD AND NOT _0108_CH1_IDD);
(*  *)
(* Rung L3 *)
IF NOT %ML2600.0 THEN _0109_OUTEN := 15; END_IF;
(* Rung L6 *)
IF _ON AND %IX1.1.37 THEN _t1 := 0 > _0108_CH0_DATA; END_IF;
IF _t1 THEN _0108_CH0_DATA := 0; END_IF;
(* Rung L10 *)
IF _ON AND %IX1.1.38 THEN _t2 := 0 > _0108_CH1_DATA; END_IF;
IF _t2 THEN _0108_CH1_DATA := 0; END_IF;
(* Rung L14 *)
IF _0108_CH0_ACT AND _0109_CH0_ACT AND %IX1.1.37 THEN %WW1000 := _0108_CH0_DATA; END_IF;
IF _0108_CH0_ACT AND _0109_CH0_ACT AND %IX1.1.37 AND %IX1.1.37 THEN
    _0109_CH0_DATA := _0108_CH0_DATA;
END_IF;
(* Rung L17 *)
IF _0108_CH1_ACT AND _0109_CH0_ACT AND %IX1.1.38 THEN %WW1000 := _0108_CH1_DATA; END_IF;
IF _0108_CH1_ACT AND _0109_CH0_ACT AND %IX1.1.38 AND %IX1.1.38 THEN
    _0109_CH0_DATA := _0108_CH1_DATA;
END_IF;
(* DF-1 출하 유량 INOUT PUT *)
(* [#FIT] DF-1 *)
(* Rung L22 *)
%ML2600.1 := NOT (NOT _0108_CH2_IDD AND NOT _0108_CH3_IDD);
(* DF-1 CH2 PIT2 IN PUT *)
(* Rung L23 *)
IF _ON AND %IX1.1.39 THEN _t3 := 0 > _0108_CH2_DATA; END_IF;
IF _t3 THEN _0108_CH2_DATA := 0; END_IF;
(* Rung L27 *)
IF _ON AND %IX1.1.40 THEN _t4 := 0 > _0108_CH3_DATA; END_IF;
IF _t4 THEN _0108_CH3_DATA := 0; END_IF;

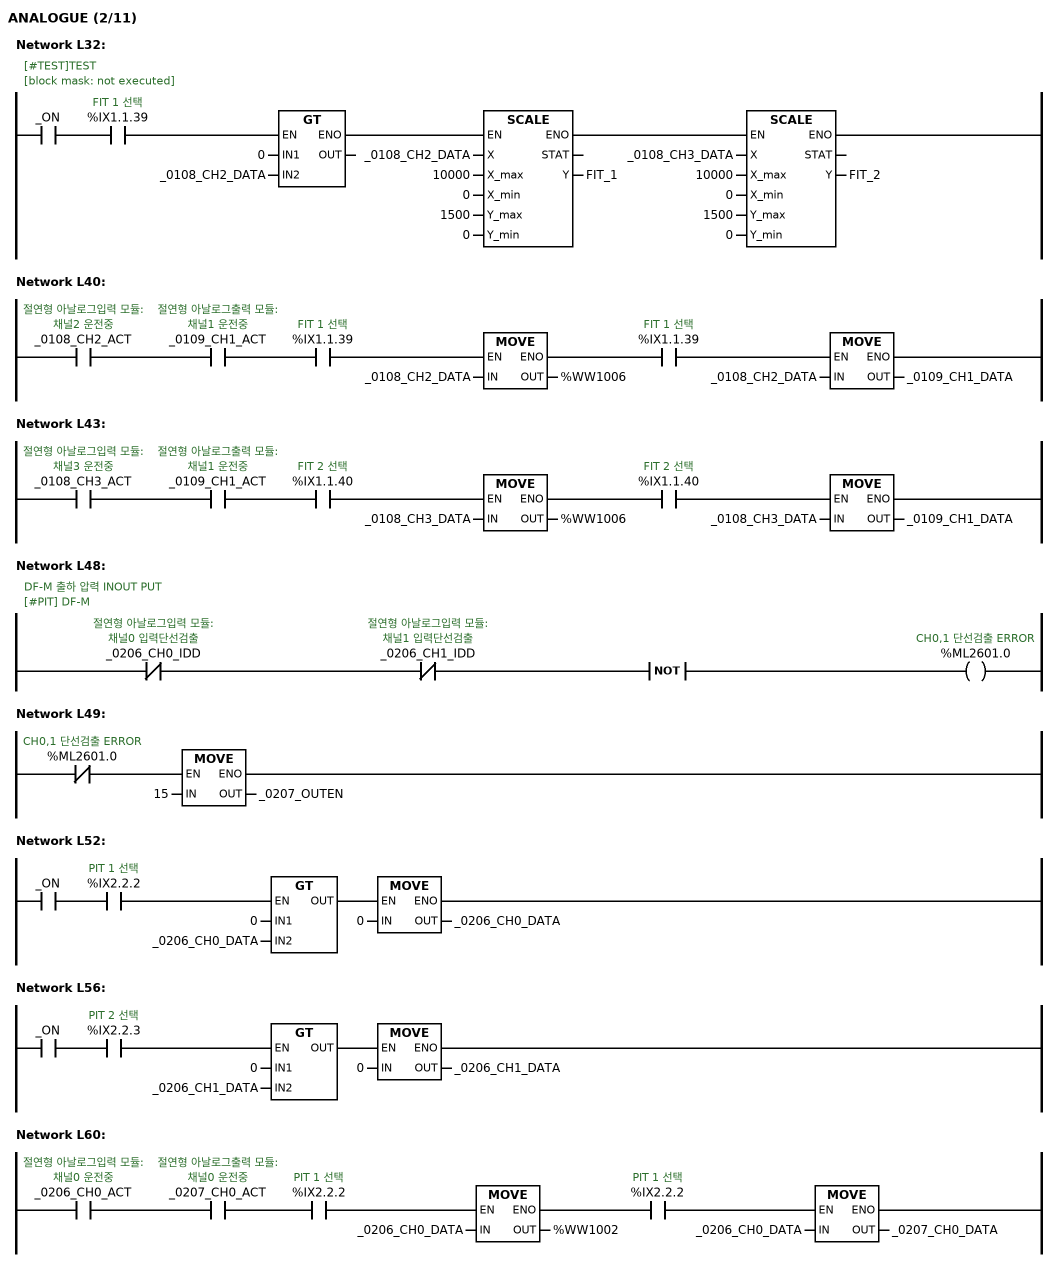
(* [#TEST]TEST *)
(* Rung L32 is block-masked: not executed *)
// IF _ON AND %IX1.1.39 THEN
//     _t5 := 0 > _0108_CH2_DATA;
//     SCALE(X := _0108_CH2_DATA, X_max := 10000, X_min := 0, Y_max := 1500, Y_min := 0, Y => FIT_1);
//     SCALE(X := _0108_CH3_DATA, X_max := 10000, X_min := 0, Y_max := 1500, Y_min := 0, Y => FIT_2);
// END_IF;
(*  *)
(* Rung L40 *)
IF _0108_CH2_ACT AND _0109_CH1_ACT AND %IX1.1.39 THEN %WW1006 := _0108_CH2_DATA; END_IF;
IF _0108_CH2_ACT AND _0109_CH1_ACT AND %IX1.1.39 AND %IX1.1.39 THEN
    _0109_CH1_DATA := _0108_CH2_DATA;
END_IF;
(* Rung L43 *)
IF _0108_CH3_ACT AND _0109_CH1_ACT AND %IX1.1.40 THEN %WW1006 := _0108_CH3_DATA; END_IF;
IF _0108_CH3_ACT AND _0109_CH1_ACT AND %IX1.1.40 AND %IX1.1.40 THEN
    _0109_CH1_DATA := _0108_CH3_DATA;
END_IF;
(* DF-M 출하 압력 INOUT PUT *)
(* [#PIT] DF-M *)
(* Rung L48 *)
%ML2601.0 := NOT (NOT _0206_CH0_IDD AND NOT _0206_CH1_IDD);
(*  *)
(* Rung L49 *)
IF NOT %ML2601.0 THEN _0207_OUTEN := 15; END_IF;
(* Rung L52 *)
IF _ON AND %IX2.2.2 THEN _t6 := 0 > _0206_CH0_DATA; END_IF;
IF _t6 THEN _0206_CH0_DATA := 0; END_IF;
(* Rung L56 *)
IF _ON AND %IX2.2.3 THEN _t7 := 0 > _0206_CH1_DATA; END_IF;
IF _t7 THEN _0206_CH1_DATA := 0; END_IF;
(* Rung L60 *)
IF _0206_CH0_ACT AND _0207_CH0_ACT AND %IX2.2.2 THEN %WW1002 := _0206_CH0_DATA; END_IF;
IF _0206_CH0_ACT AND _0207_CH0_ACT AND %IX2.2.2 AND %IX2.2.2 THEN
    _0207_CH0_DATA := _0206_CH0_DATA;
END_IF;

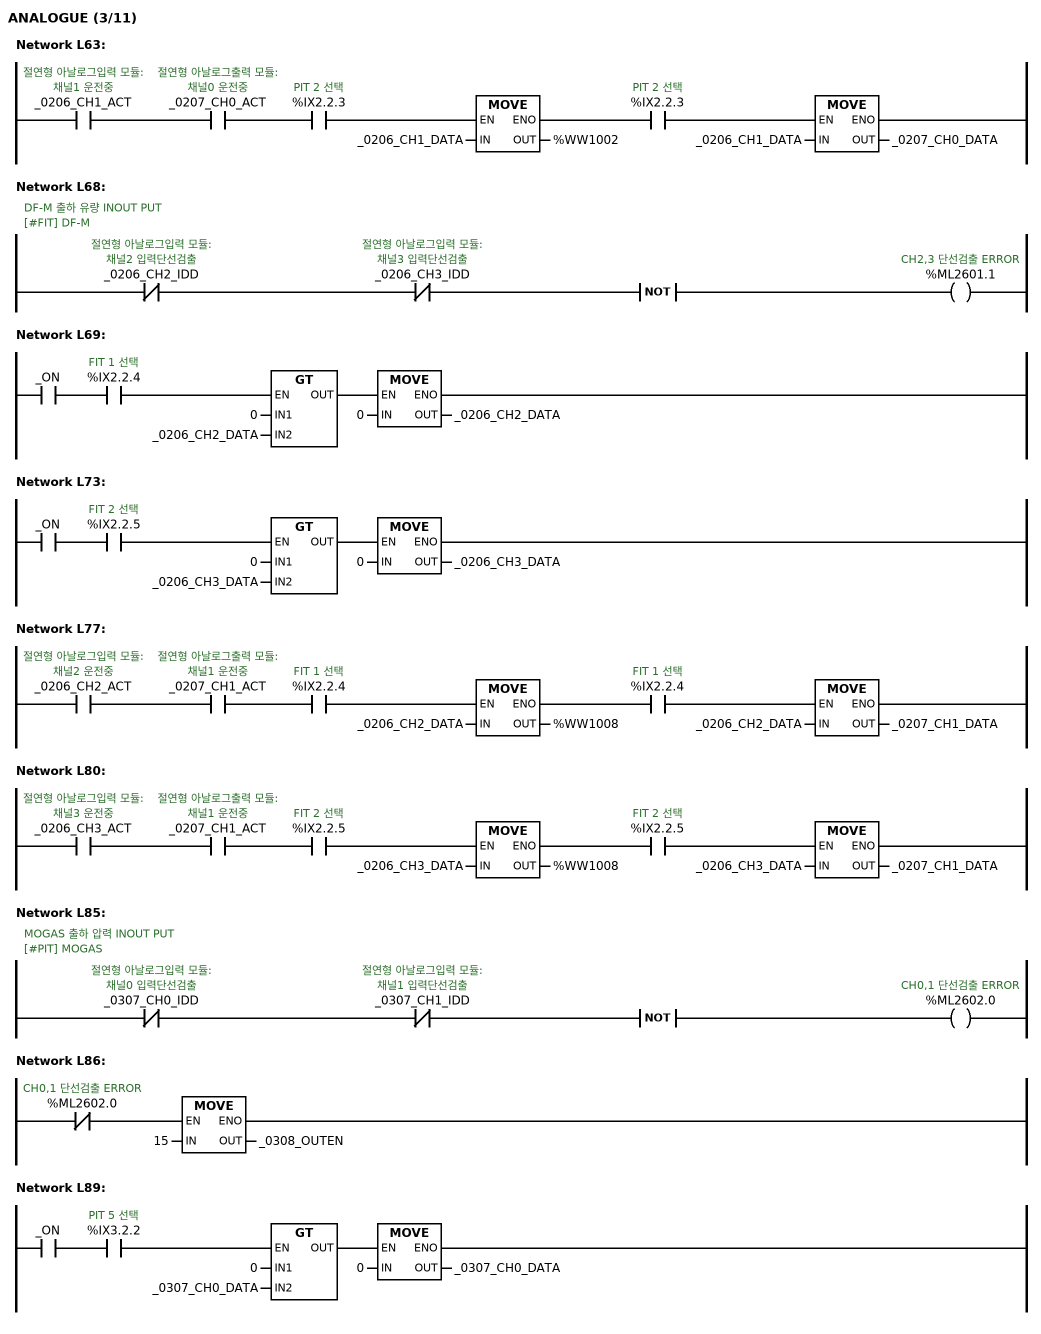
(* Rung L63 *)
IF _0206_CH1_ACT AND _0207_CH0_ACT AND %IX2.2.3 THEN %WW1002 := _0206_CH1_DATA; END_IF;
IF _0206_CH1_ACT AND _0207_CH0_ACT AND %IX2.2.3 AND %IX2.2.3 THEN
    _0207_CH0_DATA := _0206_CH1_DATA;
END_IF;
(* DF-M 출하 유량 INOUT PUT *)
(* [#FIT] DF-M *)
(* Rung L68 *)
%ML2601.1 := NOT (NOT _0206_CH2_IDD AND NOT _0206_CH3_IDD);
(*  *)
(* Rung L69 *)
IF _ON AND %IX2.2.4 THEN _t8 := 0 > _0206_CH2_DATA; END_IF;
IF _t8 THEN _0206_CH2_DATA := 0; END_IF;
(* Rung L73 *)
IF _ON AND %IX2.2.5 THEN _t9 := 0 > _0206_CH3_DATA; END_IF;
IF _t9 THEN _0206_CH3_DATA := 0; END_IF;
(* Rung L77 *)
IF _0206_CH2_ACT AND _0207_CH1_ACT AND %IX2.2.4 THEN %WW1008 := _0206_CH2_DATA; END_IF;
IF _0206_CH2_ACT AND _0207_CH1_ACT AND %IX2.2.4 AND %IX2.2.4 THEN
    _0207_CH1_DATA := _0206_CH2_DATA;
END_IF;
(* Rung L80 *)
IF _0206_CH3_ACT AND _0207_CH1_ACT AND %IX2.2.5 THEN %WW1008 := _0206_CH3_DATA; END_IF;
IF _0206_CH3_ACT AND _0207_CH1_ACT AND %IX2.2.5 AND %IX2.2.5 THEN
    _0207_CH1_DATA := _0206_CH3_DATA;
END_IF;
(* MOGAS 출하 압력 INOUT PUT *)
(* [#PIT] MOGAS *)
(* Rung L85 *)
%ML2602.0 := NOT (NOT _0307_CH0_IDD AND NOT _0307_CH1_IDD);
(*  *)
(* Rung L86 *)
IF NOT %ML2602.0 THEN _0308_OUTEN := 15; END_IF;
(* Rung L89 *)
IF _ON AND %IX3.2.2 THEN _t10 := 0 > _0307_CH0_DATA; END_IF;
IF _t10 THEN _0307_CH0_DATA := 0; END_IF;

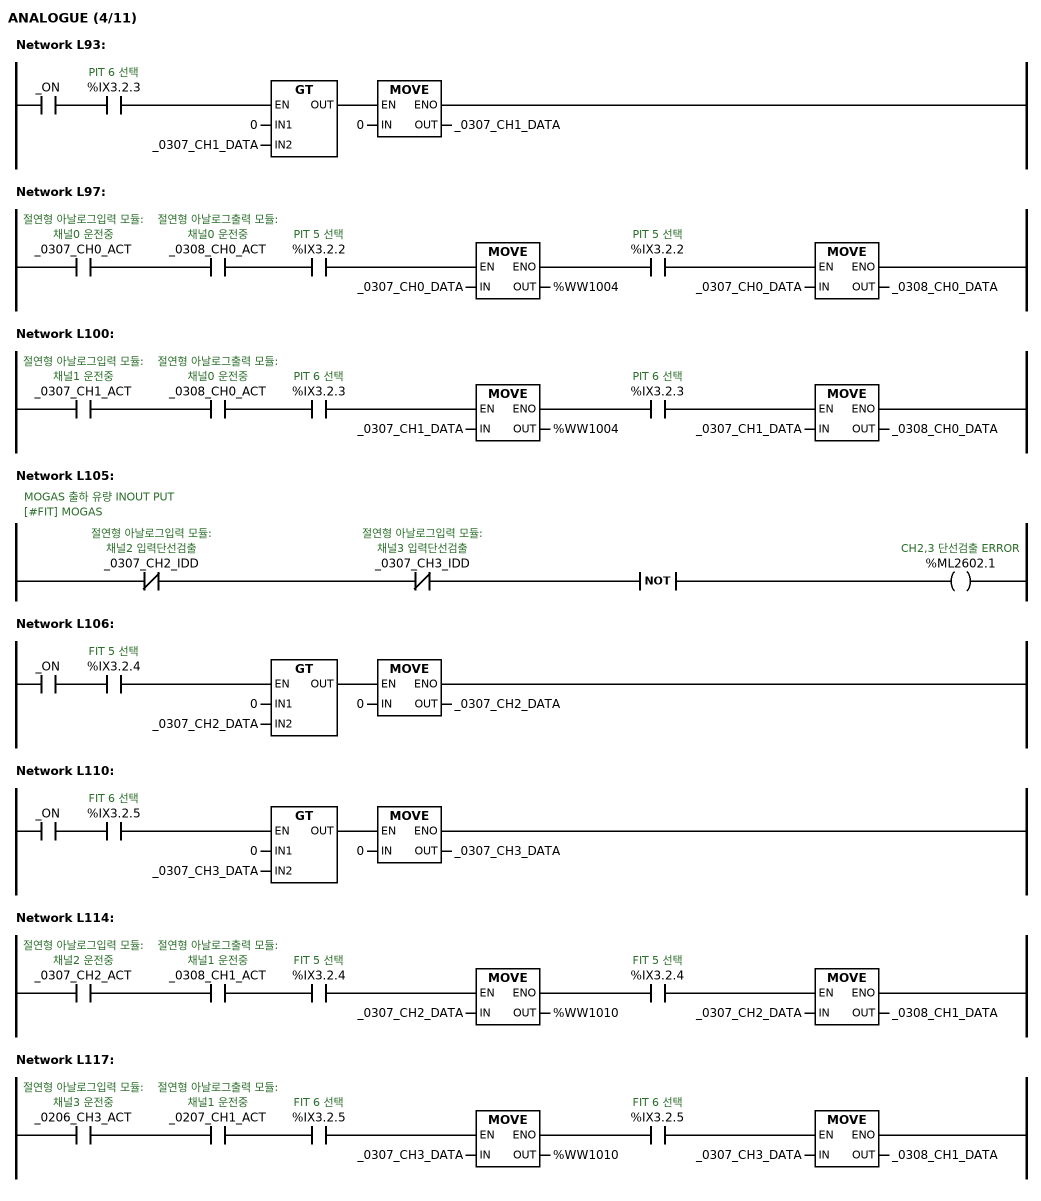
(* Rung L93 *)
IF _ON AND %IX3.2.3 THEN _t11 := 0 > _0307_CH1_DATA; END_IF;
IF _t11 THEN _0307_CH1_DATA := 0; END_IF;
(* Rung L97 *)
IF _0307_CH0_ACT AND _0308_CH0_ACT AND %IX3.2.2 THEN %WW1004 := _0307_CH0_DATA; END_IF;
IF _0307_CH0_ACT AND _0308_CH0_ACT AND %IX3.2.2 AND %IX3.2.2 THEN
    _0308_CH0_DATA := _0307_CH0_DATA;
END_IF;
(* Rung L100 *)
IF _0307_CH1_ACT AND _0308_CH0_ACT AND %IX3.2.3 THEN %WW1004 := _0307_CH1_DATA; END_IF;
IF _0307_CH1_ACT AND _0308_CH0_ACT AND %IX3.2.3 AND %IX3.2.3 THEN
    _0308_CH0_DATA := _0307_CH1_DATA;
END_IF;
(* MOGAS 출하 유량 INOUT PUT *)
(* [#FIT] MOGAS *)
(* Rung L105 *)
%ML2602.1 := NOT (NOT _0307_CH2_IDD AND NOT _0307_CH3_IDD);
(*  *)
(* Rung L106 *)
IF _ON AND %IX3.2.4 THEN _t12 := 0 > _0307_CH2_DATA; END_IF;
IF _t12 THEN _0307_CH2_DATA := 0; END_IF;
(* Rung L110 *)
IF _ON AND %IX3.2.5 THEN _t13 := 0 > _0307_CH3_DATA; END_IF;
IF _t13 THEN _0307_CH3_DATA := 0; END_IF;
(* Rung L114 *)
IF _0307_CH2_ACT AND _0308_CH1_ACT AND %IX3.2.4 THEN %WW1010 := _0307_CH2_DATA; END_IF;
IF _0307_CH2_ACT AND _0308_CH1_ACT AND %IX3.2.4 AND %IX3.2.4 THEN
    _0308_CH1_DATA := _0307_CH2_DATA;
END_IF;
(* Rung L117 *)
IF _0206_CH3_ACT AND _0207_CH1_ACT AND %IX3.2.5 THEN %WW1010 := _0307_CH3_DATA; END_IF;
IF _0206_CH3_ACT AND _0207_CH1_ACT AND %IX3.2.5 AND %IX3.2.5 THEN
    _0308_CH1_DATA := _0307_CH3_DATA;
END_IF;

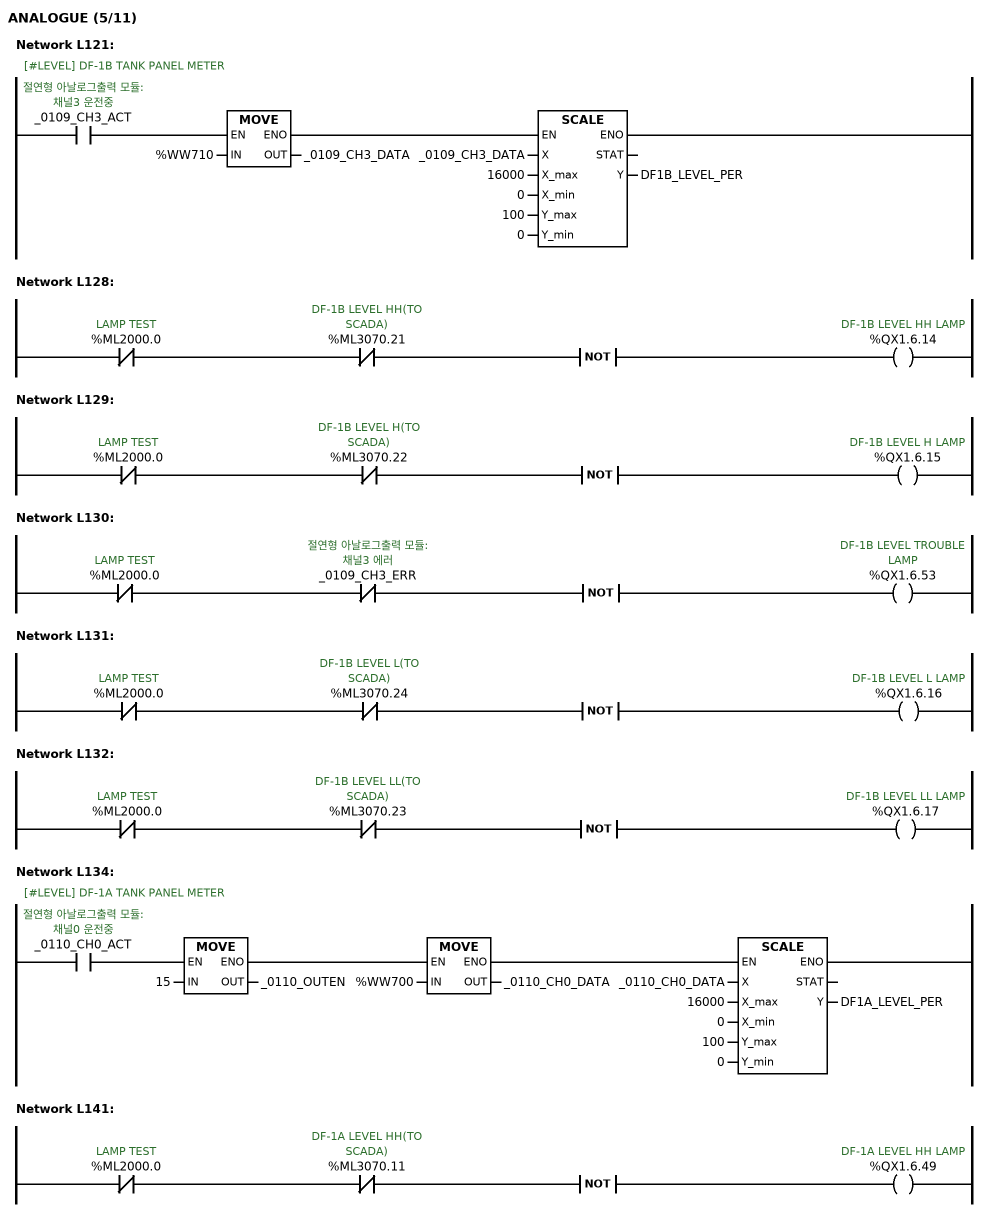
(* [#LEVEL] DF-1B TANK PANEL METER *)
(* Rung L121 *)
IF _0109_CH3_ACT THEN
    _0109_CH3_DATA := %WW710;
    SCALE(X := _0109_CH3_DATA, X_max := 16000, X_min := 0, Y_max := 100, Y_min := 0, Y => DF1B_LEVEL_PER);
END_IF;
(* Rung L128 *)
%QX1.6.14 := NOT (NOT %ML2000.0 AND NOT %ML3070.21);
(* Rung L129 *)
%QX1.6.15 := NOT (NOT %ML2000.0 AND NOT %ML3070.22);
(* Rung L130 *)
%QX1.6.53 := NOT (NOT %ML2000.0 AND NOT _0109_CH3_ERR);
(* Rung L131 *)
%QX1.6.16 := NOT (NOT %ML2000.0 AND NOT %ML3070.24);
(* Rung L132 *)
%QX1.6.17 := NOT (NOT %ML2000.0 AND NOT %ML3070.23);
(* [#LEVEL] DF-1A TANK PANEL METER *)
(* Rung L134 *)
IF _0110_CH0_ACT THEN
    _0110_OUTEN := 15;
    _0110_CH0_DATA := %WW700;
    SCALE(X := _0110_CH0_DATA, X_max := 16000, X_min := 0, Y_max := 100, Y_min := 0, Y => DF1A_LEVEL_PER);
END_IF;
(* Rung L141 *)
%QX1.6.49 := NOT (NOT %ML2000.0 AND NOT %ML3070.11);

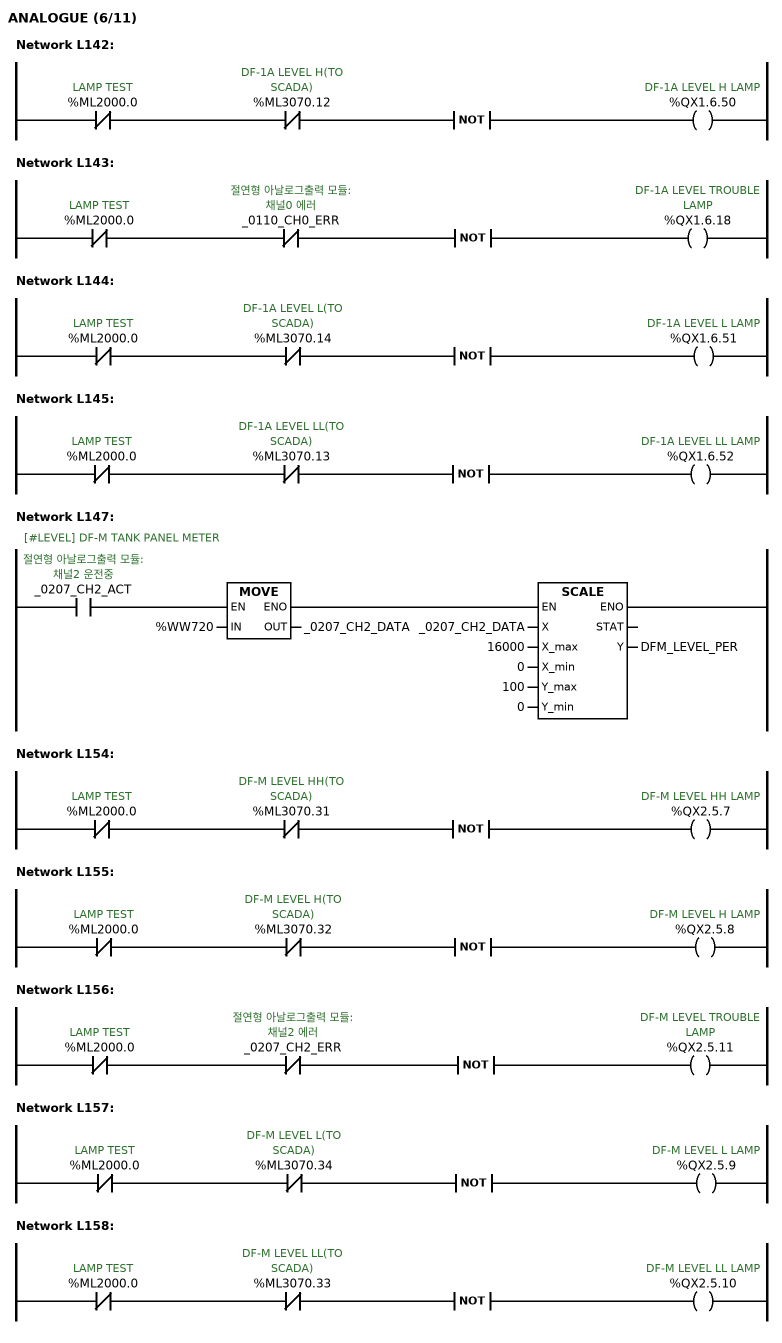
(* Rung L142 *)
%QX1.6.50 := NOT (NOT %ML2000.0 AND NOT %ML3070.12);
(* Rung L143 *)
%QX1.6.18 := NOT (NOT %ML2000.0 AND NOT _0110_CH0_ERR);
(* Rung L144 *)
%QX1.6.51 := NOT (NOT %ML2000.0 AND NOT %ML3070.14);
(* Rung L145 *)
%QX1.6.52 := NOT (NOT %ML2000.0 AND NOT %ML3070.13);
(* [#LEVEL] DF-M TANK PANEL METER *)
(* Rung L147 *)
IF _0207_CH2_ACT THEN
    _0207_CH2_DATA := %WW720;
    SCALE(X := _0207_CH2_DATA, X_max := 16000, X_min := 0, Y_max := 100, Y_min := 0, Y => DFM_LEVEL_PER);
END_IF;
(* Rung L154 *)
%QX2.5.7 := NOT (NOT %ML2000.0 AND NOT %ML3070.31);
(* Rung L155 *)
%QX2.5.8 := NOT (NOT %ML2000.0 AND NOT %ML3070.32);
(* Rung L156 *)
%QX2.5.11 := NOT (NOT %ML2000.0 AND NOT _0207_CH2_ERR);
(* Rung L157 *)
%QX2.5.9 := NOT (NOT %ML2000.0 AND NOT %ML3070.34);
(* Rung L158 *)
%QX2.5.10 := NOT (NOT %ML2000.0 AND NOT %ML3070.33);

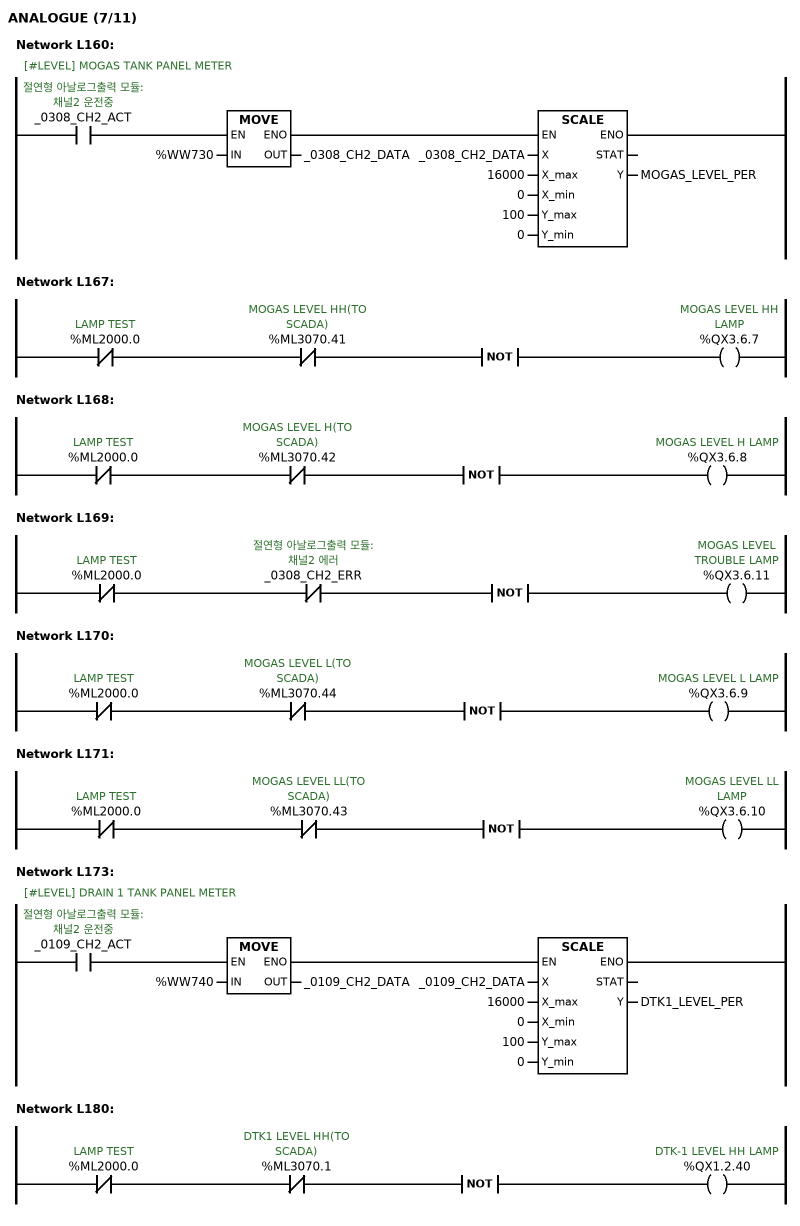
(* [#LEVEL] MOGAS TANK PANEL METER *)
(* Rung L160 *)
IF _0308_CH2_ACT THEN
    _0308_CH2_DATA := %WW730;
    SCALE(X := _0308_CH2_DATA, X_max := 16000, X_min := 0, Y_max := 100, Y_min := 0, Y => MOGAS_LEVEL_PER);
END_IF;
(* Rung L167 *)
%QX3.6.7 := NOT (NOT %ML2000.0 AND NOT %ML3070.41);
(* Rung L168 *)
%QX3.6.8 := NOT (NOT %ML2000.0 AND NOT %ML3070.42);
(* Rung L169 *)
%QX3.6.11 := NOT (NOT %ML2000.0 AND NOT _0308_CH2_ERR);
(* Rung L170 *)
%QX3.6.9 := NOT (NOT %ML2000.0 AND NOT %ML3070.44);
(* Rung L171 *)
%QX3.6.10 := NOT (NOT %ML2000.0 AND NOT %ML3070.43);
(* [#LEVEL] DRAIN 1 TANK PANEL METER *)
(* Rung L173 *)
IF _0109_CH2_ACT THEN
    _0109_CH2_DATA := %WW740;
    SCALE(X := _0109_CH2_DATA, X_max := 16000, X_min := 0, Y_max := 100, Y_min := 0, Y => DTK1_LEVEL_PER);
END_IF;
(* Rung L180 *)
%QX1.2.40 := NOT (NOT %ML2000.0 AND NOT %ML3070.1);

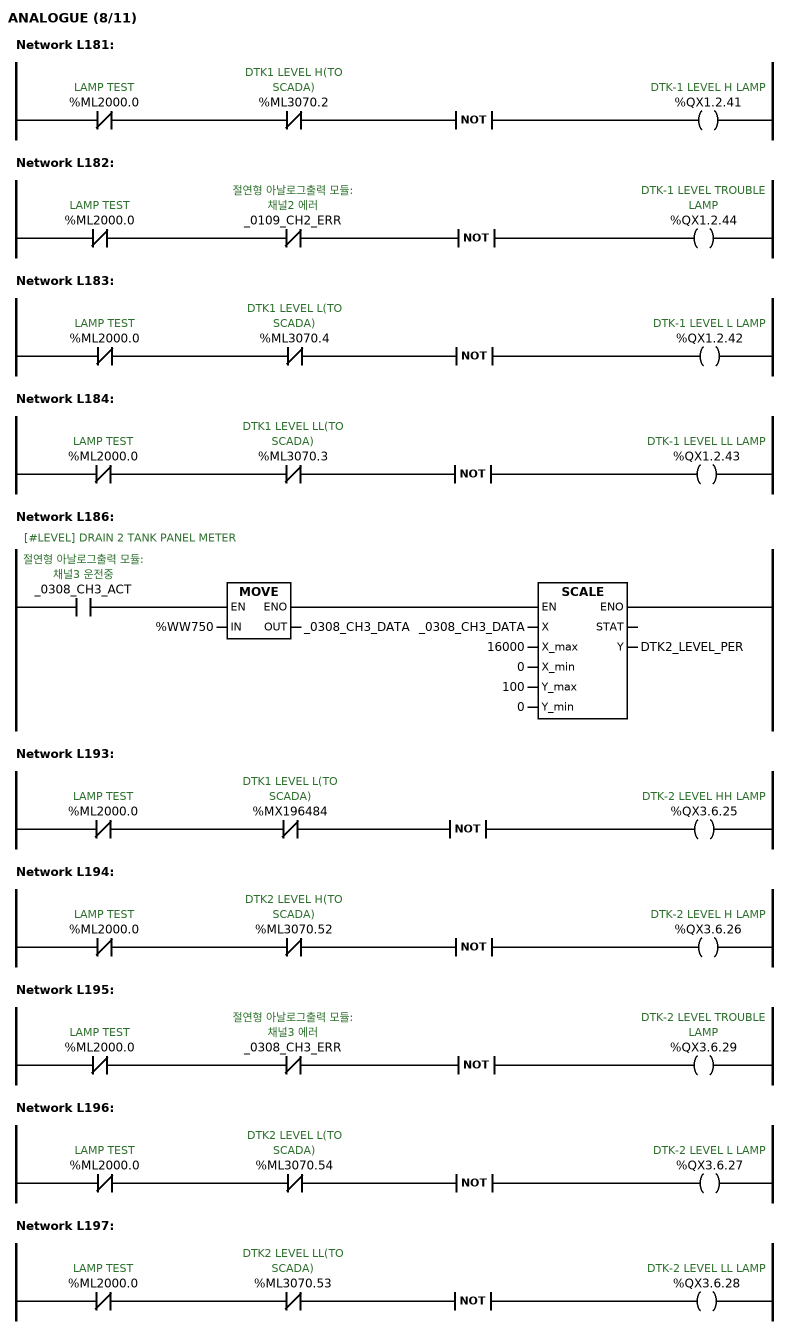
(* Rung L181 *)
%QX1.2.41 := NOT (NOT %ML2000.0 AND NOT %ML3070.2);
(* Rung L182 *)
%QX1.2.44 := NOT (NOT %ML2000.0 AND NOT _0109_CH2_ERR);
(* Rung L183 *)
%QX1.2.42 := NOT (NOT %ML2000.0 AND NOT %ML3070.4);
(* Rung L184 *)
%QX1.2.43 := NOT (NOT %ML2000.0 AND NOT %ML3070.3);
(* [#LEVEL] DRAIN 2 TANK PANEL METER *)
(* Rung L186 *)
IF _0308_CH3_ACT THEN
    _0308_CH3_DATA := %WW750;
    SCALE(X := _0308_CH3_DATA, X_max := 16000, X_min := 0, Y_max := 100, Y_min := 0, Y => DTK2_LEVEL_PER);
END_IF;
(* Rung L193 *)
%QX3.6.25 := NOT (NOT %ML2000.0 AND NOT %MX196484);
(* Rung L194 *)
%QX3.6.26 := NOT (NOT %ML2000.0 AND NOT %ML3070.52);
(* Rung L195 *)
%QX3.6.29 := NOT (NOT %ML2000.0 AND NOT _0308_CH3_ERR);
(* Rung L196 *)
%QX3.6.27 := NOT (NOT %ML2000.0 AND NOT %ML3070.54);
(* Rung L197 *)
%QX3.6.28 := NOT (NOT %ML2000.0 AND NOT %ML3070.53);

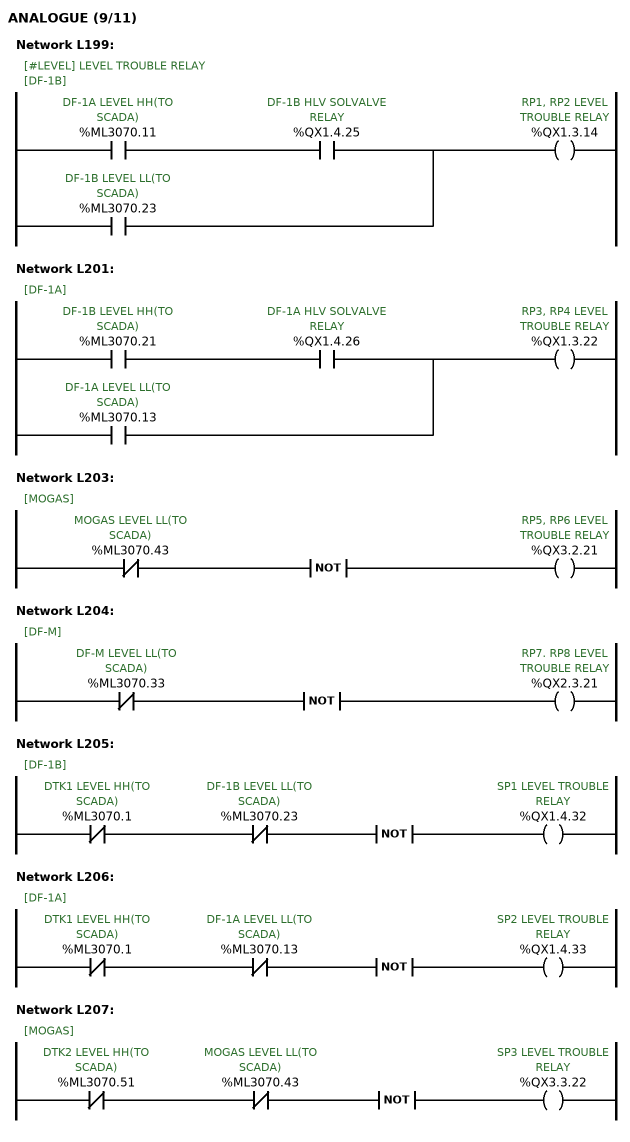
(* [#LEVEL] LEVEL TROUBLE RELAY *)
(* Rung L199 *)
%QX1.3.14 := (%ML3070.11 AND %QX1.4.25) OR %ML3070.23;
(* [DF-1B] *)
(* Rung L201 *)
%QX1.3.22 := (%ML3070.21 AND %QX1.4.26) OR %ML3070.13;
(* [DF-1A] *)
(* Rung L203 *)
%QX3.2.21 := %ML3070.43;
(* [MOGAS] *)
(* Rung L204 *)
%QX2.3.21 := %ML3070.33;
(* [DF-M] *)
(* Rung L205 *)
%QX1.4.32 := NOT (NOT %ML3070.1 AND NOT %ML3070.23);
(* [DF-1B] *)
(* Rung L206 *)
%QX1.4.33 := NOT (NOT %ML3070.1 AND NOT %ML3070.13);
(* [DF-1A] *)
(* Rung L207 *)
%QX3.3.22 := NOT (NOT %ML3070.51 AND NOT %ML3070.43);
(* [MOGAS] *)

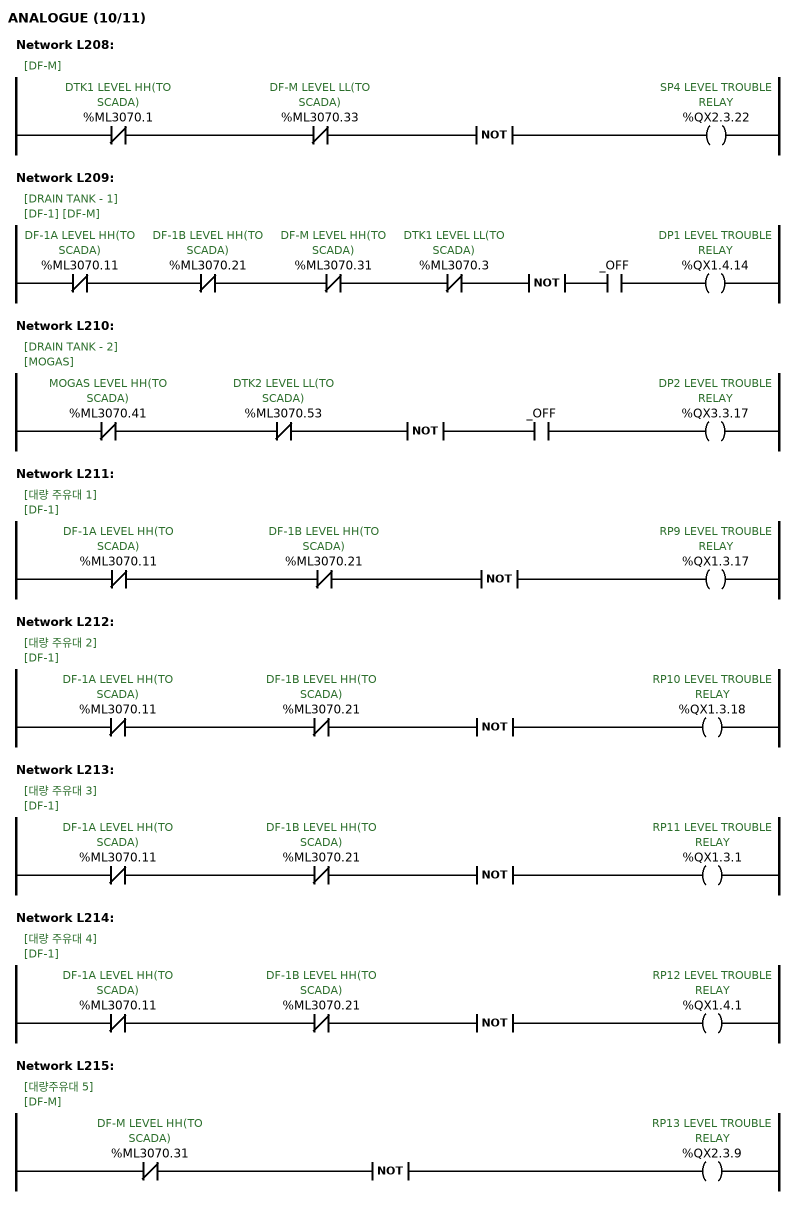
(* Rung L208 *)
%QX2.3.22 := NOT (NOT %ML3070.1 AND NOT %ML3070.33);
(* [DF-M] *)
(* Rung L209 *)
%QX1.4.14 := NOT (NOT %ML3070.11 AND NOT %ML3070.21 AND NOT %ML3070.31 AND NOT %ML3070.3) AND _OFF;
(* [DRAIN TANK - 1] / [DF-1] [DF-M] *)
(* Rung L210 *)
%QX3.3.17 := NOT (NOT %ML3070.41 AND NOT %ML3070.53) AND _OFF;
(* [DRAIN TANK - 2] / [MOGAS] *)
(* Rung L211 *)
%QX1.3.17 := NOT (NOT %ML3070.11 AND NOT %ML3070.21);
(* [대량 주유대 1] / [DF-1] *)
(* Rung L212 *)
%QX1.3.18 := NOT (NOT %ML3070.11 AND NOT %ML3070.21);
(* [대량 주유대 2] / [DF-1] *)
(* Rung L213 *)
%QX1.3.1 := NOT (NOT %ML3070.11 AND NOT %ML3070.21);
(* [대량 주유대 3] / [DF-1] *)
(* Rung L214 *)
%QX1.4.1 := NOT (NOT %ML3070.11 AND NOT %ML3070.21);
(* [대량 주유대 4] / [DF-1] *)
(* Rung L215 *)
%QX2.3.9 := %ML3070.31;
(* [대량주유대 5] / [DF-M] *)

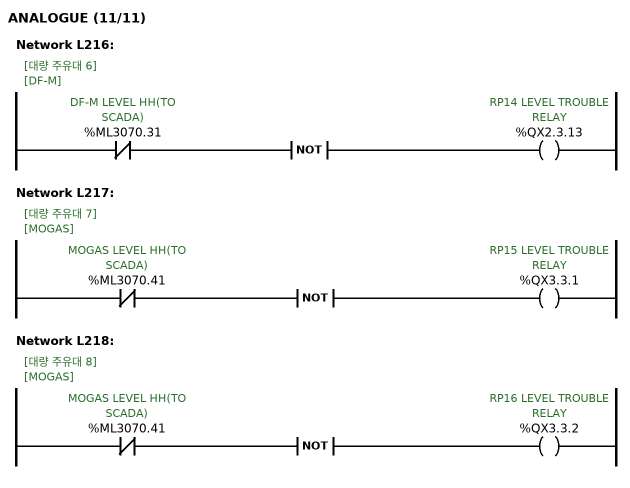
(* Rung L216 *)
%QX2.3.13 := %ML3070.31;
(* [대량 주유대 6] / [DF-M] *)
(* Rung L217 *)
%QX3.3.1 := %ML3070.41;
(* [대량 주유대 7] / [MOGAS] *)
(* Rung L218 *)
%QX3.3.2 := %ML3070.41;
(* [대량 주유대 8] / [MOGAS] *)
END_PROGRAM

PROGRAM COMMUNICATION (* task: 스캔 프로그램 *)

